		strTemp := strPath;
		strTemp := CONCAT(strTemp , aFileList[intOldestFile].sFileName);
		THIS^.M_FileDelete(strTemp);
		
		IF (uinSubStep = cSubStep_Finished) THEN
			intCmd := cFOLDER_HDL_CMD_DONE;
			uinStep := cStep_Refresh; 
		ELSIF (uinSubStep = cSubStep_Error) THEN
			intCmd := cFOLDER_HDL_CMD_DONE;
			uinStep := cStep_Error;
		END_IF
		
	cStep_Error:	
		// entry action
		IF (uinStep<>uinStep_old) THEN
			// written in sub Out_strInfo := 'Error';
			Out_bolBusy := FALSE;
			uinStep_old := uinStep;
		END_IF
		
		IF (intCmd<>cFOLDER_HDL_CMD_DONE) THEN
			Out_udiErrId := 0;
			uinSubStep := cSubStep_Done;
			uinStep := cStep_Wait4Job;
		END_IF
END_CASE

PROPERTY PUBLIC FileSupervisionPeriod : TIME
GET
FileSupervisionPeriod := timFileSupervisionPeriod;
END_GET
SET
timFileSupervisionPeriod := FileSupervisionPeriod;
END_SET
END_PROPERTY

PROPERTY PUBLIC get_FileList : ARRAY[1..cFILE_HDL_MAX_NR_OF_FILE_TO_MANAGE]  OF ST_FindFileEntry;
GET
uinSubStep := 0;

WHILE (THIS^.M_RefreshFileList()=FALSE) DO
	//wait until read all files in folder
END_WHILE

THIS^.M_SortFileList(); // sort last write date -> oldest at position 1!
END_GET
END_PROPERTY

PROPERTY get_NewestFileEntry : ST_FindFileEntry
GET
uinSubStep := 0;
(* läuft nicvht???
WHILE (THIS^.M_RefrehFileList()=FALSE) DO
	//wait until read all files in folder
END_WHILE

THIS^.M_SortFileList(); // sort last write date -> oldest at position 1!
*)
get_NewestFileEntry := aFileList[udiNrOfFilesInFolder];
END_GET
END_PROPERTY

METHOD PUBLIC M_Cmd_RefreshFileList : BOOL
intCmd := cFOLDER_HDL_CMD_REFRESH_FILE_LIST;
END_METHOD

METHOD PROTECTED M_FileDelete : BOOL
VAR_INPUT
	strPathName : T_MaxString;  
END_VAR
VAR
	strMyName : STRING := 'M_FileDelete: ';
END_VAR

CASE uinSubStep OF
	cSubStep_Done:	
		Out_strInfo :=  CONCAT(CONCAT(Out_strInfo, strMyName) , 'start');
		
		fbFileDelete_1.sNetId := strNetId;
		fbFileDelete_1.sPathName := strPathName;
		fbFileDelete_1.ePath := PATH_GENERIC;
		fbFileDelete_1.tTimeout := T#3S;
		fbFileDelete_1(bExecute:= FALSE);
		fbFileDelete_1(bExecute:= TRUE);
		
		uinSubStep := 1;
		
	1: 
		Out_strInfo :=  CONCAT(CONCAT(Out_strInfo, strMyName) , 'busy');	

		(* wait until function block not busy *)
		fbFileDelete_1( bExecute := FALSE );
		IF NOT fbFileDelete_1.bBusy THEN
			IF NOT fbFileDelete_1.bError THEN
				uinSubStep := cSubStep_Finished;
			ELSE 
				Out_udiErrId := fbFileDelete_1.nErrID;
				uinSubStep := cSubStep_Error;
			END_IF
		END_IF
		
	cSubStep_Finished: 
		// succesfully finished
		
	cSubStep_Error:
		Out_strInfo :=  CONCAT(CONCAT(Out_strInfo, strMyName) , CONCAT('error active - number:' , DWORD_TO_HEXSTR( fbFileDelete_1.nErrID, 0, FALSE )));
		Out_udiErrId := fbFileDelete_1.nErrID;
END_CASE
END_METHOD

METHOD PUBLIC M_FileExist : BOOL
VAR_INPUT
	strPathName : Tc2_System.T_MaxString;
END_VAR
VAR
	fbEnum : FB_EnumFindFileEntry := ( sNetID := '', tTimeout := T#5S, sPathName := strPathName );
	uinState : UINT:=0;
END_VAR
WHILE (uinState<>10) DO
	CASE uinState OF
	0:
		fbEnum.sNetId := strNetId;
		fbEnum.eCmd := eEnumCmd_First; (* enum first entry *)
		uinState := 1;
	
	1: (* enum one entry *)
		fbEnum( bExecute := FALSE );
		fbEnum( bExecute := TRUE );
		uinState := 2;
	
	2: (* wait until function block not busy *)
		fbEnum( bExecute := FALSE );
		IF NOT fbEnum.bBusy THEN
			IF NOT fbEnum.bError THEN
				IF NOT fbEnum.bEOE THEN
					M_FileExist := TRUE;
					EXIT;
				ELSE (* no more entries *)
					M_FileExist := FALSE;
					EXIT;
				END_IF
			ELSE (* log error *)
				M_FileExist := FALSE;
				EXIT;
			END_IF
		END_IF
	END_CASE
END_WHILE
END_METHOD

METHOD M_getFileInfo : ST_FindFileEntry
VAR_INPUT
	IN_strFileNameWithExt : Tc2_System.T_MaxString;// Contains the filename with extension
END_VAR
VAR
	ii : UDINT;
	udiUpperLimit : UDINT;
END_VAR
IF (udiNrOfFilesInFolder<cFILE_HDL_MAX_NR_OF_FILE_TO_MANAGE) THEN
	udiUpperLimit := udiNrOfFilesInFolder;
ELSE
	udiUpperLimit := cFILE_HDL_MAX_NR_OF_FILE_TO_MANAGE;	
END_IF

FOR ii:= 0 TO udiUpperLimit DO
	IF (FIND(aFileList[ii].sFileName,IN_strFileNameWithExt)<>0) THEN
		M_getFileInfo := aFileList[ii];
		EXIT;
	END_IF
END_FOR
END_METHOD

METHOD PUBLIC M_GetFileSize : LREAL
VAR_INPUT
	In_strFileName: T_MaxString;
END_VAR
VAR
	i:UDINT;
END_VAR
IF (udiNrOfFilesInFolder=0) THEN
	WHILE (THIS^.M_RefreshFileList()=FALSE) DO
		//wait until read all files in folder
	END_WHILE
END_IF

M_GetFileSize := 0.0;

FOR i := 1 TO udiNrOfFilesInFolder BY 1 DO
	IF (In_strFileName = aFileList[i].sFileName) THEN
		M_GetFileSize := Tc2_Utilities.UINT64_TO_LREAL(aFileList[i].fileSize);
		EXIT;
	END_IF
END_FOR;
END_METHOD

METHOD PUBLIC M_Init : BOOL
VAR_INPUT
	IN_strPath : Tc2_System.T_MaxString; 	// Contains only the path 
	IN_strPrefixFileName : Tc2_System.T_MaxString;// Contains only the filename
	IN_strFileExt : Tc2_System.T_MaxString;	// Contains only the ext
	In_strNetId: STRING(23); // NetId to write to foreign system drives
END_VAR
VAR
	strTemp: Tc2_System.T_MaxString;
END_VAR
strNetId := In_strNetId;
strPath := IN_strPath;
strFilePrefix := IN_strPrefixFileName;
strFileExt := IN_strFileExt;
strTemp := strPath;//todo check path allready added / CONCAT(strPath , '\');
strTemp := CONCAT(strTemp , strFilePrefix);
IF (strFileExt='') THEN
	strPathName := strTemp;
ELSE
	strTemp := CONCAT(strTemp , '.');
	strPathName := CONCAT(strTemp , strFileExt);
END_IF
uinStep := 0;
bolInitDone := TRUE;
END_METHOD

METHOD PUBLIC M_RefreshFileList : BOOL
VAR
	strMyName : STRING := 'M_RefrehFileList: ';
	strTemp : STRING;
END_VAR
CASE uinSubStep OF
	cSubStep_Done:	
		Out_strInfo :=  CONCAT(CONCAT(Out_strInfo, strMyName) , 'start');
		
		M_RefreshFileList := FALSE;
		udiNrOfFilesInFolder := 0;
		
		// define proberties for searching files in folder
		fbEnumFindFileList_1.sNetId := strNetId;

		strTemp := strPath;//todo check path allready added / CONCAT(strPath , '\');
		strTemp := CONCAT(strTemp , strFilePrefix);
		IF (strFileExt='') THEN
			strTemp := CONCAT(strTemp , '*'); // all data types
		ELSE
			strTemp := CONCAT(strTemp , '*.');
			strTemp := CONCAT(strTemp , strFileExt);
		END_IF

		fbEnumFindFileList_1.sPathName := strTemp; // read all files in the defined folder with the defined extension
        fbEnumFindFileList_1.pFindList := ADR(aFileList);
        fbEnumFindFileList_1.cbFindList := SIZEOF(aFileList);
        fbEnumFindFileList_1.tTimeout := DEFAULT_ADS_TIMEOUT;
		fbEnumFindFileList_1.eCmd := E_EnumCmdType.eEnumCmd_First;	(* enum first entry *)
		uinSubStep := 1;
		
	1: 
		Out_strInfo :=  CONCAT(CONCAT(Out_strInfo, strMyName) , 'Reading files in folder busy');	
		
		(* enum one entry *)
		IF bolAbort THEN
			bolAbort := FALSE;
			fbEnumFindFileList_1.eCmd := E_EnumCmdType.eEnumCmd_Abort;
		END_IF
		
		fbEnumFindFileList_1( bExecute := FALSE );
		fbEnumFindFileList_1( bExecute := TRUE );
		uinSubStep := 2;
		
	2:	
		Out_strInfo := CONCAT(CONCAT(Out_strInfo, strMyName) , 'Reading files in folder busy');	
		
		(* wait until function block not busy *)
		fbEnumFindFileList_1( bExecute := FALSE );
		IF NOT fbEnumFindFileList_1.bBusy THEN
			udiNrOfFilesInFolder := fbEnumFindFileList_1.nFindFiles;
			IF NOT fbEnumFindFileList_1.bError THEN
				IF NOT fbEnumFindFileList_1.bEOE THEN
					bolFileNrExceedArraySize := TRUE;
					(* read more informations -> not meaningful 
					fbEnumFindFileList_1.eCmd := E_EnumCmdType.eEnumCmd_Next; (* enum next entry *)
					uinSubStep := 1;*)
					uinSubStep := cSubStep_Finished; // reduce maximum in cyclic actions...-> delete if > max 
				ELSE (* no more entries *)
					uinSubStep := cSubStep_Finished;
				END_IF
			ELSE (* log error *)
				Out_udiErrId := fbEnumFindFileList_1.nErrID;
				uinSubStep := cSubStep_Error;
			END_IF
		END_IF

	cSubStep_Finished: 
		// succesfully finished
		M_RefreshFileList := TRUE;
	cSubStep_Error:
		Out_strInfo :=  CONCAT(CONCAT(Out_strInfo, strMyName) , CONCAT('error active - number:' , DWORD_TO_HEXSTR( fbEnumFindFileList_1.nErrID, 0, FALSE )));
		Out_udiErrId := fbEnumFindFileList_1.nErrID;
		M_RefreshFileList := TRUE;
END_CASE
END_METHOD

METHOD PUBLIC M_SortFileList : BOOL
VAR_INPUT

END_VAR
VAR
	stTempFile 	: ST_FindFileEntry;
	bolNoChangeDone: BOOL;
	i,j :UDINT;
END_VAR
// BubbleSort
M_SortFileList := FALSE;

IF (udiNrOfFilesInFolder>1) THEN
	lreTotalFileSize := UINT64_TO_LREAL(aFileList[1].fileSize);
	FOR i := 1 TO udiNrOfFilesInFolder BY 1 DO
		bolNoChangeDone := TRUE;
		FOR j := 1 TO (udiNrOfFilesInFolder-i) BY 1 DO
			IF (i=1) THEN// count total filesize
				lreTotalFileSize := lreTotalFileSize + Tc2_Utilities.UINT64_TO_LREAL(aFileList[j+1].fileSize);
			END_IF
			
			IF (FILETIME_TO_DT(aFileList[j].lastWriteTime) > FILETIME_TO_DT(aFileList[j + 1].lastWriteTime)) THEN
				// swap files
				memcpy(ADR(stTempFile), ADR(aFileList[j]),SIZEOF(stTempFile));
				memcpy(ADR(aFileList[j]), ADR(aFileList[j + 1]),SIZEOF(stTempFile));
				memcpy(ADR(aFileList[j + 1]), ADR(stTempFile),SIZEOF(stTempFile));
				bolNoChangeDone := FALSE; // at least one change done
			END_IF
			
		END_FOR; 
		IF (bolNoChangeDone) THEN
			EXIT;
		END_IF
	END_FOR;
END_IF;
M_SortFileList := TRUE;
END_METHOD

PROPERTY MaxNrOfFilesInFolder : UINT
GET
MaxNrOfFilesInFolder := uinMaxNrOfFilesInFolder;
END_GET
SET
// not more files allowed as defined in struct....Sort problem
IF (MaxNrOfFilesInFolder<cFILE_HDL_MAX_NR_OF_FILE_TO_MANAGE) THEN
	uinMaxNrOfFilesInFolder := MaxNrOfFilesInFolder;
ELSE
	uinMaxNrOfFilesInFolder := UDINT_TO_UINT(cFILE_HDL_MAX_NR_OF_FILE_TO_MANAGE-1);	
END_IF
END_SET
END_PROPERTY

END_FUNCTION_BLOCK

// POUs/Utility/GHT [Generic Hash Table]/FB_GHT
FUNCTION_BLOCK FB_GHT IMPLEMENTS IGHT
VAR CONSTANT
	MAX_HASH_LISTS: INT := 3;
	MAX_HASHLIST_ENTRIES: INT := 50;
	CUTOFF_A: ULINT := 4000000000;
	CUTOFF_B: ULINT := 8000000000;
END_VAR
VAR
	m_bolDeleteItems: BOOL;
	m_uintCount: UINT;
	m_fbHashTable: ARRAY[0..(MAX_HASH_LISTS - 1)] OF FB_HashTableCtrl;
	m_hHashTable: ARRAY[0..(MAX_HASH_LISTS - 1)] OF T_HHASHTABLE;
	m_uliCutoff: ARRAY[0..(MAX_HASH_LISTS - 1)] OF ULINT;
	m_aHashTableBuffer: ARRAY[0..(MAX_HASH_LISTS - 1)] OF T_GHTHashTableBuffer;
END_VAR

{attribute 'object_name' := 'AddItem'}
METHOD AddItem : BOOL
VAR_INPUT
	uliKey: ULINT;
	pData: POINTER TO BYTE;
END_VAR
VAR
	iIdx: INT;
END_VAR
iIdx := GetTableIdx(uliKey);

m_fbHashTable[iIdx].A_Add( key := ULINT_TO_UDINT(uliKey-m_uliCutoff[iIdx]), putValue := pData, hTable := m_hHashTable[iIdx] );

IF m_fbHashTable[iIdx].bOk THEN
	m_uintCount := m_uintCount + 1;
END_IF
END_METHOD

{attribute 'object_name' := 'Clear'}
METHOD Clear : BOOL
VAR_INPUT
	bolFreePointer: BOOL;
END_VAR
VAR
	iIdx: INT;
	pData: POINTER TO BYTE;
END_VAR
FOR iIdx := 0 TO MAX_HASH_LISTS - 1 DO
	IF bolFreePointer THEN
		m_fbHashTable[iIdx].A_GetFirst(hTable := m_hHashTable[iIdx]);

		WHILE m_fbHashTable[iIdx].bOk DO
			pData := m_fbHashTable[iIdx].getValue;
			__DELETE(pData);
			m_fbHashTable[iIdx].A_GetNext(hTable := m_hHashTable[iIdx]);
		END_WHILE
		
	END_IF
	
	m_fbHashTable[iIdx].A_RemoveAll(hTable := m_hHashTable[iIdx]);
END_FOR

m_uintCount := 0;
END_METHOD

PROPERTY Count : UINT
GET
END_GET
END_PROPERTY

{attribute 'object_name' := 'FB_init'}
METHOD FB_init : BOOL
VAR_INPUT
	/// if TRUE, the retain variables are initialized (warm start / cold start)
	bInitRetains: BOOL;
	/// if TRUE, the instance afterwards gets moved into the copy code (online change)
	bInCopyCode: BOOL;
END_VAR
m_uliCutoff[0] := 0;
m_uliCutoff[1] := CUTOFF_A;
m_uliCutoff[2] := CUTOFF_B;

m_uintCount := 0;
END_METHOD

{attribute 'object_name' := 'GetTableIdx'}
METHOD PRIVATE GetTableIdx : INT
VAR_INPUT
	uliBarcode: ULINT;
END_VAR
IF uliBarcode < CUTOFF_A THEN
	GetTableIdx := 0;
	RETURN;
END_IF

IF uliBarcode > CUTOFF_B THEN
	GetTableIdx := 2;
	RETURN;
END_IF

GetTableIdx := 1;
END_METHOD

{attribute 'object_name' := 'Initialize'}
METHOD Initialize : BOOL
F_CreateHashTableHnd( ADR( m_aHashTableBuffer[0].aBuffer ), SIZEOF( m_aHashTableBuffer[0].aBuffer ), m_hHashTable[0] );
F_CreateHashTableHnd( ADR( m_aHashTableBuffer[1].aBuffer ), SIZEOF( m_aHashTableBuffer[1].aBuffer ), m_hHashTable[1] );
F_CreateHashTableHnd( ADR( m_aHashTableBuffer[2].aBuffer ), SIZEOF( m_aHashTableBuffer[2].aBuffer ), m_hHashTable[2] );
END_METHOD

{attribute 'object_name' := 'Lookup'}
METHOD Lookup : POINTER TO BYTE
VAR_INPUT
	uliKey: ULINT;
	bolRemove: BOOL;
END_VAR
VAR
	pfbHashTable: POINTER TO FB_HashTableCtrl;
	phHashTable: POINTER TO T_HHASHTABLE;
	uliCutoff: ULINT;
	iIdx: INT;
END_VAR
iIdx := GetTableIdx(uliKey);

m_fbHashTable[iIdx].A_Lookup( key := ULINT_TO_UDINT(uliKey-m_uliCutoff[iIdx]), hTable := m_hHashTable[iIdx] );

IF m_fbHashTable[iIdx].bOk THEN
	Lookup := m_fbHashTable[iIdx].getValue;
	
	IF bolRemove THEN
		m_fbHashTable[iIdx].A_Remove( key := ULINT_TO_UDINT(uliKey-m_uliCutoff[iIdx]), hTable := m_hHashTable[iIdx]);

		IF m_fbHashTable[iIdx].bOk THEN
			m_uintCount := m_uintCount - 1;
		END_IF
	END_IF
ELSE
	Lookup := NULL;
END_IF
END_METHOD

END_FUNCTION_BLOCK

// POUs/Utility/GHT [Generic Hash Table]/IGHT
INTERFACE IGHT

{attribute 'object_name' := 'AddItem'}
METHOD AddItem : BOOL
VAR_INPUT
	uliKey: ULINT;
	pData: POINTER TO BYTE;
END_VAR
END_METHOD

{attribute 'object_name' := 'Clear'}
METHOD Clear : BOOL
VAR_INPUT
	bolFreePointer: BOOL;
END_VAR
END_METHOD

PROPERTY Count : UINT
GET
END_GET
END_PROPERTY

{attribute 'object_name' := 'Initialize'}
METHOD Initialize : BOOL
END_METHOD

{attribute 'object_name' := 'Lookup'}
METHOD Lookup : POINTER TO BYTE
VAR_INPUT
	uliKey: ULINT;
	bolRemove: BOOL;
END_VAR
END_METHOD

END_INTERFACE

// POUs/Utility/Logger/BasLog/FB_BasLogTest_Client
FUNCTION_BLOCK FB_BasLogTest_Client
VAR_INPUT
	In_p_fbBasLog: POINTER TO FB_BasLog; // only one central FB_BasLog instance allowed per PLC!!!
END_VAR
VAR_OUTPUT
END_VAR
VAR
	stData : T_Bl_BaseStruc;
	bolInit : BOOL := FALSE;
	pReadHandle : POINTER TO POINTER TO T_Queue_Info;
	uinInitStatus : UINT;
	uinChangeMaskStatus :UINT;
	uinReadStatus : UINT;
	bolChangeMask : BOOL;
	bolRead : BOOL;
	fbTimeStamp: FB_TimeStamp;
END_VAR

(*__________________________________________________________________________________________________
¦	
¦	Vistaprint Schweiz GmbH
¦	CH - 8401 Winterthur
¦
¦	www.vistaprint.ch - info@vistaprint.ch
¦___________________________________________________________________________________________________

Function desription:
Example and test programm for testing the base log system - read data from base log

History:
Version		Date			Author		Comment
---------------------------------------------------------------------------------------------------
0.00.1		14.07.2014		AVME/KVO	Start history
___________________________________________________________________________________________________*)

// system init onetime after start up
IF (bolInit=FALSE) THEN
	// init timer system
	fbTimeStamp.In_strNetId := ''; // use local system time
	fbTimeStamp.In_t_CycleTimeRefreshTimeZone := T#15M; // cyclic check time zone settings
	//init baselog system, one time should be called per baslog system
	In_p_fbBasLog^.M_ClientInit(In_strClientName:='BaseLog',In_udiMask := 16#FFFFFFFF, In_uinNrOfElement:= 128,In_p_fbTimeStamp:=ADR(fbTimeStamp),In_bolUseLocalTimeStamp:=TRUE,Out_pHandle=>pReadHandle,Out_uinStatus=>uinInitStatus);
	
	bolInit := TRUE;
END_IF

fbTimeStamp(); // cyclic call needed for valid time stamp / synchronisation
	
(* change mak on runtime *)
IF (bolRead = TRUE) THEN
	(* cyclically read out of data*)
	uinReadStatus:= In_p_fbBasLog^.M_Read(In_pHandle:=pReadHandle,In_pData:=ADR(stData)); 
END_IF

(* change mask on runtime *)
IF (bolChangeMask = TRUE) THEN
	uinChangeMaskStatus := In_p_fbBasLog^.M_ChangeMask(In_strClientName:='BaseLog',In_udiNewMask:= 16#0F0F0F0F);
	bolChangeMask := FALSE;
END_IF

END_FUNCTION_BLOCK

// POUs/Utility/Logger/BasLog/FB_BasLogTest_Sender
FUNCTION_BLOCK FB_BasLogTest_Sender
VAR_INPUT
	In_p_fbBasLog: POINTER TO FB_BasLog; // only one central FB_BasLog instance allowed per PLC!!!
END_VAR
VAR_OUTPUT
END_VAR
VAR
	bolInit : BOOL := FALSE;
	pHandle : POINTER TO T_Bl_LibHandleRow;
	uinGetHandleStatus : UINT;
	uinWriteStatus :UINT;
	uinDoWrite : UINT;
	dinPar1 : DINT;
	strText1 : STRING(30):='Controller 1';
	strText2 : STRING(30):='Alarm sub info';
END_VAR

(*__________________________________________________________________________________________________
¦	
¦	Vistaprint Schweiz GmbH
¦	CH - 8401 Winterthur
¦
¦	www.vistaprint.ch - info@vistaprint.ch
¦___________________________________________________________________________________________________

Function desription:
Example and test programm for testing the queue system - write data to base log

History:
Version		Date			Author		Comment
---------------------------------------------------------------------------------------------------
0.00.1		14.07.2014		AVME/KVO	Start history
___________________________________________________________________________________________________*)

// system init onetime after start up
IF (bolInit=FALSE) THEN
	uinGetHandleStatus := In_p_fbBasLog^.M_GetHandle(Out_pHandle=>pHandle);
	
	bolInit := TRUE;
END_IF

// write base log entries
IF (uinDoWrite>0) THEN
	uinDoWrite := uinDoWrite - 1;
	dinPar1 := dinPar1 + 1;
	uinWriteStatus := In_p_fbBasLog^.M_Log(In_pHandle:=pHandle,In_udiLogType:=BasLog.cLOGTYPE_ALARM,In_intCtrlID:=11,In_strText1:=strText1,In_strText2:=strText2,In_dinPar1:=dinPar1,In_dinPar2:=0,In_dinPar3:=0,In_dinPar4:=0) ;
END_IF

END_FUNCTION_BLOCK

// POUs/Utility/Logger/DatLog/FB_DatLog
FUNCTION_BLOCK FB_DatLog
VAR_INPUT
END_VAR
VAR_OUTPUT
END_VAR
VAR
	stDatLogLibInfo : T_DL_LibInfo;
	fbPLC_ReadSymInfo: PLC_ReadSymInfoByNameEx; // only one init allowed on the same time....
END_VAR

(*__________________________________________________________________________________________________
¦	
¦	Vistaprint Schweiz GmbH
¦	CH - 8401 Winterthur
¦
¦	www.vistaprint.ch - info@vistaprint.ch
¦___________________________________________________________________________________________________

Function desription:
Base logger system. The FUB must be called defined globally one time in PLC-program. After that the implemented 
sender and receiver must interact over the public methodes of the FB_BasLog.

History:
Version		Date			Author		Comment
---------------------------------------------------------------------------------------------------
0.00.1		14.07.2014		AVME/KVO	Start history
___________________________________________________________________________________________________*)

METHOD PROTECTED M_AllocMEM : POINTER TO BYTE

VAR_INPUT
	In_SizeOfBuffer : UINT; // Byte size of quee to allocate
END_VAR
// Debug counter
M_AllocMEM := __NEW(BYTE,In_SizeOfBuffer);

// check if allocate memory is ok
IF (M_AllocMEM=TC3_MEMMAN.NULL) THEN
	M_AllocMEM := TC3_MEMMAN.NULL;
ELSE
	Tc2_System.MEMSET(M_AllocMEM,0,In_SizeOfBuffer); // init with zero.
END_IF
END_METHOD

METHOD PRIVATE M_CheckAndAppendDatLogInfo : Pointer TO T_DL_SysInfo
VAR_INPUT
	In_strDatLogName: STRING(DatLog.cMAX_SYS_NAME_LENGTH); // name of the client
END_VAR
VAR
	pstSysInfo: POINTER TO T_DL_SysInfo;
END_VAR
// methode check, if data log allready exists and if not allocate a new system
// -> return reference on new system

// exist at least one data log system
IF (stDatLogLibInfo.pstDatLogSysInfo=TC3_MEMMAN.NULL) THEN
	// create  a new system
	stDatLogLibInfo.pstDatLogSysInfo := M_AllocMEM(SIZEOF(T_DL_SysInfo));

	IF (stDatLogLibInfo.pstDatLogSysInfo=TC3_MEMMAN.NULL) THEN
		M_CheckAndAppendDatLogInfo := TC3_MEMMAN.NULL;
		RETURN;
	END_IF
	
	// data log name entry in info system
	stDatLogLibInfo.pstDatLogSysInfo^.strDatLogName := In_strDatLogName;
	M_CheckAndAppendDatLogInfo := stDatLogLibInfo.pstDatLogSysInfo;
	RETURN;
END_IF

// after this point the system has to exist
IF (stDatLogLibInfo.pstDatLogSysInfo<>TC3_MEMMAN.NULL) THEN
	pstSysInfo := stDatLogLibInfo.pstDatLogSysInfo;
	
	WHILE (pstSysInfo<>TC3_MEMMAN.NULL) DO
		IF (pstSysInfo^.strDatLogName=In_strDatLogName) THEN
			// data log name found -> return handle
			M_CheckAndAppendDatLogInfo := pstSysInfo;
			RETURN;
		END_IF
		
		// last element
		IF (pstSysInfo^.pstNextDatLogSystem=TC3_MEMMAN.NULL) THEN
			// the requested log name does not exist -> allocate a new one
			pstSysInfo^.pstNextDatLogSystem := M_AllocMEM(SIZEOF(T_DL_SysInfo));

			IF (pstSysInfo^.pstNextDatLogSystem<>TC3_MEMMAN.NULL) THEN
				pstSysInfo := pstSysInfo^.pstNextDatLogSystem;
				// data log name entry in info system
				pstSysInfo^.strDatLogName := In_strDatLogName;
				M_CheckAndAppendDatLogInfo := pstSysInfo;
				RETURN;
			ELSE
				M_CheckAndAppendDatLogInfo := TC3_MEMMAN.NULL;
				RETURN;
			END_IF
		ELSE
			// reference next
			pstSysInfo := pstSysInfo^.pstNextDatLogSystem;
		END_IF
	END_WHILE
END_IF
END_METHOD

METHOD PUBLIC M_GetHandle : UINT
VAR_INPUT
	In_strDatLogName: STRING(DatLog.cMAX_SYS_NAME_LENGTH); // name of the client
	In_p_fbBasLog: POINTER TO FB_BasLog; // only one central FB_BasLog instance allowed per PLC!!!
END_VAR
VAR_OUTPUT
	Out_pHandle : POINTER TO BYTE; // handle of log system for write (M_Log)
	Out_udiStatus : UDINT; //0 => successful done, <>0 => error
END_VAR
VAR
	pstSysInfo: POINTER TO T_DL_SysInfo;
	uinGetHandleStatus : UINT;
END_VAR

// check if log system allready exists or not, if not allocate a new one
	pstSysInfo := M_CheckAndAppendDatLogInfo(In_strDatLogName:=In_strDatLogName);
	IF (pstSysInfo=TC3_MEMMAN.NULL) THEN
		Out_udiStatus := DatLog.cERR_MEM_ALLOC;
		RETURN;
	END_IF
	
	// log on base log system
	uinGetHandleStatus := In_p_fbBasLog^.M_GetHandle(Out_pHandle=>pstSysInfo^.pBaseLogHandle);
	
	// check error
	IF (uinGetHandleStatus<>0) THEN
		Out_udiStatus := UINT_TO_UDINT(uinGetHandleStatus);
		RETURN;
	ELSE
		pstSysInfo^.p_fbBasLog := In_p_fbBasLog;
		Out_pHandle := pstSysInfo;
	END_IF
END_METHOD

METHOD PUBLIC M_Init : BOOL
VAR_INPUT
	In_bolExecute : BOOL;
	In_strDatLogName: STRING(DatLog.cMAX_SYS_NAME_LENGTH); // name of the client
	In_a_strDataDefinition: ARRAY[0..DatLog.cMAX_NR_OF_VAR] OF STRING(DatLog.cMAX_VAR_NAME_LEN); // complete VarName: p.e.:MAIN.INIT_TASK.VARINT
	In_uinStartId: UINT;	// Start ident for item index -> cfg file config has to match with this number!
	In_Port : T_AmsPort;	// on plc the first runtime system is the 801, 811 ...
END_VAR
VAR_OUTPUT
	Out_udiStatus: UDINT;		 // 0 => successful done, <>0 => error
	Out_bolDone: BOOL;			// Done
END_VAR
VAR
	pstSysInfo: POINTER TO T_DL_SysInfo;
	pstItem : POINTER TO T_DL_Item;
	ii : UINT;
END_VAR

IF (In_bolExecute=TRUE) THEN
	// check if log system allready exists or not, if not allocate a new one
	pstSysInfo := M_CheckAndAppendDatLogInfo(In_strDatLogName:=In_strDatLogName);
	IF (pstSysInfo=TC3_MEMMAN.NULL) THEN
		Out_udiStatus := DatLog.cERR_MEM_ALLOC;
		RETURN;
	END_IF

	IF (stDatLogLibInfo.stStatemachine.bolExecute_old=FALSE) THEN // reset statemachine
		stDatLogLibInfo.stStatemachine.uinState := 1;
		Out_bolDone := FALSE;
		Out_udiStatus := 0;
		stDatLogLibInfo.stStatemachine.usiInitDone := 0;
	END_IF

CASE stDatLogLibInfo.stStatemachine.uinState OF
	1:
		//check number of elements
		FOR ii :=0 TO DatLog.cMAX_NR_OF_VAR BY 1 DO
			IF (In_a_strDataDefinition[ii]='') THEN
				EXIT;
			END_IF
		END_FOR
		
		pstSysInfo^.uinNbrOfItems := ii;
		pstSysInfo^.uinStartId := In_uinStartId;
		
		// allocate memory for items
		pstSysInfo^.pstItems := M_AllocMEM((pstSysInfo^.uinNbrOfItems*SIZEOF(T_DL_Item)));
		IF (pstSysInfo^.pstItems =TC3_MEMMAN.NULL) THEN
			Out_udiStatus := DatLog.cERR_MEM_ALLOC;
			RETURN;
		END_IF
		pstSysInfo^.uinCntReadItems := 0;
		pstSysInfo^.uinItemOffset := 0;
		stDatLogLibInfo.stStatemachine.uinState := stDatLogLibInfo.stStatemachine.uinState + 1;
		
	2:	
		fbPLC_ReadSymInfo.NETID:=''; // local PLC
		IF (In_Port=0) THEN// access first runtime system
			fbPLC_ReadSymInfo.PORT := 851;
		ELSE
			fbPLC_ReadSymInfo.PORT := In_Port;
		END_IF
		fbPLC_ReadSymInfo.SYMNAME := In_a_strDataDefinition[pstSysInfo^.uinCntReadItems];
		fbPLC_ReadSymInfo.START := FALSE;
		fbPLC_ReadSymInfo();
		fbPLC_ReadSymInfo.START := TRUE;
		fbPLC_ReadSymInfo();
		stDatLogLibInfo.stStatemachine.uinState := stDatLogLibInfo.stStatemachine.uinState + 1;
		
	3:
		fbPLC_ReadSymInfo();
		IF (fbPLC_ReadSymInfo.BUSY=FALSE) THEN
			stDatLogLibInfo.stStatemachine.uinState := stDatLogLibInfo.stStatemachine.uinState + 1;
		END_IF
		
	4:
		pstItem := pstSysInfo^.pstItems;
		IF (fbPLC_ReadSymInfo.ERR=FALSE) THEN
			pstItem[pstSysInfo^.uinCntReadItems].strPvName := In_a_strDataDefinition[pstSysInfo^.uinCntReadItems];
			pstItem[pstSysInfo^.uinCntReadItems].uinItemOffset := pstSysInfo^.uinItemOffset;
			pstItem[pstSysInfo^.uinCntReadItems].SymInfo := fbPLC_ReadSymInfo.SYMINFO;
			pstSysInfo^.uinItemOffset := pstSysInfo^.uinItemOffset + UDINT_TO_UINT(pstItem[pstSysInfo^.uinCntReadItems].SymInfo.byteSize); // offset for next
			
			// check if type ok/allowed
			IF (pstItem[pstSysInfo^.uinCntReadItems].SymInfo.symDataType = 'BOOL') THEN 
				pstItem[pstSysInfo^.uinCntReadItems].udiItemType := DatLog.cVAR_TYPE_BOOL;
			ELSIF (pstItem[pstSysInfo^.uinCntReadItems].SymInfo.symDataType = 'SINT') THEN 
				pstItem[pstSysInfo^.uinCntReadItems].udiItemType := DatLog.cVAR_TYPE_SINT;
			ELSIF (pstItem[pstSysInfo^.uinCntReadItems].SymInfo.symDataType = 'INT') THEN 
				pstItem[pstSysInfo^.uinCntReadItems].udiItemType := DatLog.cVAR_TYPE_INT;
			ELSIF (pstItem[pstSysInfo^.uinCntReadItems].SymInfo.symDataType = 'DINT') THEN 
				pstItem[pstSysInfo^.uinCntReadItems].udiItemType := DatLog.cVAR_TYPE_DINT;
			ELSIF (pstItem[pstSysInfo^.uinCntReadItems].SymInfo.symDataType = 'USINT') THEN 
				pstItem[pstSysInfo^.uinCntReadItems].udiItemType := DatLog.cVAR_TYPE_USINT;
			ELSIF (pstItem[pstSysInfo^.uinCntReadItems].SymInfo.symDataType = 'UINT') THEN 
				pstItem[pstSysInfo^.uinCntReadItems].udiItemType := DatLog.cVAR_TYPE_INT;
			ELSIF (pstItem[pstSysInfo^.uinCntReadItems].SymInfo.symDataType = 'UDINT') THEN 
				pstItem[pstSysInfo^.uinCntReadItems].udiItemType := DatLog.cVAR_TYPE_UDINT;
			ELSIF (pstItem[pstSysInfo^.uinCntReadItems].SymInfo.symDataType = 'REAL') THEN 
				pstItem[pstSysInfo^.uinCntReadItems].udiItemType := DatLog.cVAR_TYPE_REAL;
			ELSIF (FIND(STR1:=pstItem[pstSysInfo^.uinCntReadItems].SymInfo.symDataType,STR2:='STRING')<>0) THEN 
				IF (pstItem[pstSysInfo^.uinCntReadItems].SymInfo.byteSize < BasLog.cMAX_CHAR_TEXT2) THEN
					pstItem[pstSysInfo^.uinCntReadItems].udiItemType := DatLog.cVAR_TYPE_STRING;
				ELSE
					Out_udiStatus := DatLog.cERR_UNSUPPORTED_TYPE_STRING_TOO_LONG;
					RETURN;
				END_IF
			ELSE
				Out_udiStatus := DatLog.cERR_UNSUPPORTED_TYPE;
				RETURN;
			END_IF
		ELSE
			Out_udiStatus := fbPLC_ReadSymInfo.ERRID;
			RETURN;
		END_IF
		
		pstSysInfo^.uinCntReadItems := pstSysInfo^.uinCntReadItems  + 1;
		IF (pstSysInfo^.uinCntReadItems<pstSysInfo^.uinNbrOfItems) THEN // read next value
			stDatLogLibInfo.stStatemachine.uinState := 2;
		ELSE
			stDatLogLibInfo.stStatemachine.uinState := stDatLogLibInfo.stStatemachine.uinState + 1; // all items found
		END_IF
	5:
		Out_bolDone := TRUE;
		Out_udiStatus := 0;
		pstSysInfo^.usiInitOk := 1; 
END_CASE
END_IF
stDatLogLibInfo.stStatemachine.bolExecute_old := In_bolExecute;
END_METHOD

METHOD PUBLIC M_Log : UINT
VAR_INPUT
	In_pHandle : POINTER TO BYTE;// handle of log system for write (M_Log)
	In_a_pData: ARRAY [0..DatLog.cMAX_NR_OF_VAR] OF POINTER TO BYTE;// address of structure elements
END_VAR
VAR_OUTPUT
	Out_udiStatus: UDINT;		// 0 => successful done, <>0 => error
END_VAR
VAR
	pstSysInfo: POINTER TO T_DL_SysInfo;
	pstItem : POINTER TO T_DL_Item;
	pstItemEle : T_DL_Item;
	ii : UINT;
	strText2: STRING(BasLog.cMAX_CHAR_TEXT2); // informationtext2
	dinPar2 : DINT;
	dinId : DINT;
	uinStatus : UINT;
END_VAR
// check handle ok
IF (In_pHandle=TC3_MEMMAN.NULL) THEN
	M_Log := DatLog.cERR_NO_HANDLE;
	RETURN;
END_IF

// check data
IF (In_a_pData[0]=TC3_MEMMAN.NULL) THEN
	M_Log := DatLog.cERR_NO_DATE;
	RETURN;
END_IF

// access data loggger system info
pstSysInfo := In_pHandle;

// check if init ok
IF (pstSysInfo^.usiInitOk=0) THEN
	M_Log := DatLog.cERR_INIT_FAILED;
	RETURN;
END_IF

// check if items
IF (pstSysInfo^.pstItems=TC3_MEMMAN.NULL) OR (pstSysInfo^.uinNbrOfItems<=0) THEN
	M_Log := DatLog.cERR_NO_ITEMS;
	RETURN;
END_IF
// access item definitions
pstItem := pstSysInfo^.pstItems;

// inc. record id: important the id is inc bevor and after writing of data -> to be sure that no second write is done (MUTEX)
stDatLogLibInfo.udiCommonRecIdx := stDatLogLibInfo.udiCommonRecIdx + 1;
IF (stDatLogLibInfo.udiCommonRecIdx=0) THEN
	stDatLogLibInfo.udiCommonRecIdx := stDatLogLibInfo.udiCommonRecIdx + 1;
END_IF
// write record start
// AE_BL_VAR_TYPE_CMD_NEW_REC
uinStatus := pstSysInfo^.p_fbBasLog^.M_Log(In_pHandle := pstSysInfo^.pBaseLogHandle,In_udiLogType:=BasLog.cLOGTYPE_DATA,In_intCtrlID:=DatLog.cCTRL_ID,In_strText1:='DataLog',In_strText2:='AE_BL_VAR_TYPE_CMD_NEW_REC',In_dinPar1:=0,In_dinPar2:=0,In_dinPar3:=BasLog.cVAR_TYPE_CMD_NEW_REC,In_dinPar4:=UDINT_TO_DINT(stDatLogLibInfo.udiCommonRecIdx));
IF (uinStatus<>0) THEN
	M_Log := uinStatus;
	RETURN;
END_IF

// loop over all items and write data to logger
FOR ii :=0 TO (pstSysInfo^.uinNbrOfItems-1) BY 1 DO
	// write item
	pstItemEle := pstItem[ii]; // for debugging
	// id
	dinId := UINT_TO_DINT(pstSysInfo^.uinStartId + ii);
	IF (pstItem[ii].udiItemType=DatLog.cVAR_TYPE_STRING) THEN
		MEMSET(destAddr:=ADR(strText2),fillByte:=0,n:= SIZEOF(strText2)); // to be sure that a zero is at the end
		// doesn't work with beckhoff...MEMCPY(destAddr := ADR(strText2),srcAddr:= (In_pAdrData + pstItem[ii].uinItemOffset),n:=pstItem[ii].SymInfo.byteSize);
		MEMCPY(destAddr := ADR(strText2),srcAddr:= In_a_pData[ii],n:=pstItem[ii].SymInfo.byteSize);
		dinPar2 := 0;
	ELSE
		strText2 := pstItem[ii].strPvName; // just for info
		MEMCPY(destAddr := ADR(dinPar2),srcAddr:= In_a_pData[ii],n:=pstItem[ii].SymInfo.byteSize);
	END_IF
	
	// log item
	uinStatus := pstSysInfo^.p_fbBasLog^.M_Log(In_pHandle := pstSysInfo^.pBaseLogHandle,In_udiLogType:=BasLog.cLOGTYPE_DATA,In_intCtrlID:=DatLog.cCTRL_ID,In_strText1:='DataLog',In_strText2:=strText2,In_dinPar1:=dinId,In_dinPar2:=dinPar2,In_dinPar3:=UDINT_TO_DINT(pstItem[ii].udiItemType),In_dinPar4:=UDINT_TO_DINT(stDatLogLibInfo.udiCommonRecIdx));

	IF (uinStatus<>0) THEN // no stop write error number
		M_Log := uinStatus;
	END_IF
END_FOR

// write record stop
// AE_BL_VAR_TYPE_CMD_NEW_REC
uinStatus := pstSysInfo^.p_fbBasLog^.M_Log(In_pHandle := pstSysInfo^.pBaseLogHandle,In_udiLogType:=BasLog.cLOGTYPE_DATA,In_intCtrlID:=DatLog.cCTRL_ID,In_strText1:='DataLog',In_strText2:='AE_BL_VAR_TYPE_CMD_END_REC',In_dinPar1:=0,In_dinPar2:=0,In_dinPar3:=BasLog.cVAR_TYPE_CMD_END_REC,In_dinPar4:=UDINT_TO_DINT(stDatLogLibInfo.udiCommonRecIdx));
IF (uinStatus<>0) THEN
	M_Log := uinStatus;
	RETURN;
END_IF

// increment id a second time
stDatLogLibInfo.udiCommonRecIdx := stDatLogLibInfo.udiCommonRecIdx + 1;
IF (stDatLogLibInfo.udiCommonRecIdx=0) THEN
	stDatLogLibInfo.udiCommonRecIdx := stDatLogLibInfo.udiCommonRecIdx + 1;
END_IF
END_METHOD

END_FUNCTION_BLOCK

// POUs/Utility/Logger/DatLog/FB_DatLogTest_Sender
FUNCTION_BLOCK FB_DatLogTest_Sender
VAR_INPUT
	In_p_fbBasLog: POINTER TO FB_BasLog; // only one central FB_BasLog instance allowed per PLC!!!
	In_a_pData: ARRAY [0..DatLog.cMAX_NR_OF_VAR] OF POINTER TO BYTE;
	In_strTaskName: STRING(20);
	In_strValueNameOfData: STRING(20);
END_VAR
VAR_OUTPUT
	Out_bolInit : BOOL := FALSE;
END_VAR
VAR
	bolDone : BOOL;
	pDL_Handle: POINTER TO T_DL_SysInfo;
	udiStatusInit :UDINT;
	udiStatus : UDINT;
	fbDatLog: FB_DatLog;
	a_strDataDefinition :ARRAY[0..DatLog.cMAX_NR_OF_VAR] OF STRING(DatLog.cMAX_VAR_NAME_LEN);
	uinDoLogData : UINT;
	strTemp: T_MaxString;
	strTemp2: T_MaxString;
	ii : UINT;
END_VAR

(*__________________________________________________________________________________________________
¦	
¦	Vistaprint Schweiz GmbH
¦	CH - 8401 Winterthur
¦
¦	www.vistaprint.ch - info@vistaprint.ch
¦___________________________________________________________________________________________________

Function desription:
Example and test programm for testing the data logger system - write data to data log

History:
Version		Date			Author		Comment
---------------------------------------------------------------------------------------------------
0.00.1		02.09.2014		AVME/KVO	Start history
___________________________________________________________________________________________________*)

// system init onetime after start up
IF (Out_bolInit=FALSE) THEN
	
	// TODO :parse a struct on PLC...
	FOR ii := 0 TO DatLog.cMAX_NR_OF_VAR DO
		strTemp := In_strTaskName;
		strTemp := CONCAT(STR1 := strTemp,'.');
		strTemp := CONCAT(STR1 := strTemp,In_strValueNameOfData);
		strTemp := CONCAT(STR1 := strTemp,'.');
		// fillup variable elements of struct, order is important!!!!!!!!!!!!!!!!!!!!
		CASE ii OF
			0:
				strTemp2 := 'bolOk';
			1:
				strTemp2 := 'intCnt';
			2:
				strTemp2 := 'strNewText';
		ELSE
			EXIT;
		END_CASE
		a_strDataDefinition[ii] := CONCAT(STR1 := strTemp,STR2:=strTemp2);
	END_FOR
	
	fbDatLog.M_Init(In_bolExecute := TRUE,In_strDatLogName:= 'DatLog',In_a_strDataDefinition:=a_strDataDefinition,In_Port:=851,In_uinStartId:=100,Out_udiStatus=>udiStatusInit,Out_bolDone=>bolDone);
	IF (bolDone OR (udiStatusInit<>0)) THEN
		fbDatLog.M_Init(In_bolExecute := FALSE,In_strDatLogName:= 'DatLog',In_a_strDataDefinition:=a_strDataDefinition,In_Port:=851,In_uinStartId:=100); // reset statemachine
	
		IF (udiStatusInit=0) THEN
			udiStatusInit := fbDatLog.M_GetHandle(In_strDatLogName:='DatLog',In_p_fbBasLog:=In_p_fbBasLog,Out_pHandle=>pDL_Handle,Out_udiStatus=>udiStatusInit);
		END_IF
		
		Out_bolInit := TRUE;
	END_IF

ELSE
	fbDatLog.M_Init(In_bolExecute := FALSE,In_strDatLogName:= 'DatLog',In_a_strDataDefinition:=a_strDataDefinition,In_Port:=851,In_uinStartId:=100); // reset statemachine
	
END_IF

// write entry data 
IF ((pDL_Handle<>TC3_MEMMAN.NULL) AND (udiStatusInit=0) AND (Out_bolInit=TRUE)) THEN
	fbDatLog.M_Log(In_pHandle:=pDL_Handle,In_a_pData:= In_a_pData,Out_udiStatus=>udiStatus);
END_IF

END_FUNCTION_BLOCK

// POUs/Utility/Logger/FileLc/FB_FileLc
FUNCTION_BLOCK FB_FileLc
VAR_INPUT
END_VAR
VAR_OUTPUT
END_VAR
VAR
	stFileLogClientLibInfo : T_FileLc_LibInfo;
	strInfo: Tc2_System.T_MaxString;	// additional debug Info
	bolExecute_old : BOOL;
END_VAR

(*__________________________________________________________________________________________________
¦	
¦	Vistaprint Schweiz GmbH
¦	CH - 8401 Winterthur
¦
¦	www.vistaprint.ch - info@vistaprint.ch
¦___________________________________________________________________________________________________

Function desription:
File client read out informations from BaseLog system and writes based on a config file the log entries to a file.

History:
Version		Date			Author		Comment
---------------------------------------------------------------------------------------------------
0.00.1		18.08.2014		AVME/KVO	Start history
___________________________________________________________________________________________________*)

METHOD PUBLIC M_Cyclic : UDINT
VAR_INPUT
	In_pHandle: POINTER TO T_FileLc_SysInfo; // handle for cyclic call
END_VAR
VAR
	pstSysInfo : POINTER TO T_FileLc_SysInfo;
 	pstItemDataList : POINTER TO T_FileLc_ItemData;
  	pstItemCfgList: POINTER TO T_FileLc_ItemCfg;
	stData : T_Bl_BaseStruc; // Data struct for read out
	uinReadStatus : UINT;
	ii : UINT;
	jj : UINT;
	bolWriteRecord : BOOL;
	pstrTmp : POINTER TO T_MaxString;
	strTmp:T_MaxString;
	p_Tmp_bytTmpFileBuffer : POINTER TO BYTE;
	bolKVO:BOOL;
	udiStatus : UDINT;
END_VAR
// check handle ok
IF (In_pHandle=TC3_MEMMAN.NULL) THEN
	M_Cyclic := FileLc.cERR_HANDLE;
	RETURN;
END_IF

// handle=SysInfo
pstSysInfo := In_pHandle;

// call time stamp asynchronous synchronisation
stFileLogClientLibInfo.fbTimeStamp();

// write data after a defined time to file
IF (pstSysInfo^.stFileHandler.udiWriteTimer<pstSysInfo^.stConfig.udiMaxTimeWriteToFile) THEN
	pstSysInfo^.stFileHandler.udiWriteTimer := pstSysInfo^.stFileHandler.udiWriteTimer + pstSysInfo^.udiCylceTimeMs; // add cycle time
ELSE
	pstSysInfo^.stFileHandler.udiWriteTimer := 0; // reset timer
	pstSysInfo^.stFileHandler.usiCmd := FileLc.cCMD_FLUSHBUF; // write entries to file
END_IF

// call file handler
M_Cyclic := pstSysInfo^.stFileHandler.FB_FileLc_FileHdl.M_Cyclic(In_pstSysInfo:=pstSysInfo);

(* ------------------------------------------------------------------------
Baselog buffer read out
--------------------------------------------------------------------------*)
//20 perhaps dynamic define over Level????
IF (pstSysInfo^.stItemInfo.uinActNbrOfItems>0) THEN
	FOR ii := 0 TO ((pstSysInfo^.stItemInfo.uinActNbrOfItems-1) * 20) BY 1 DO
		// Move record buffer to file buffer
		IF ((pstSysInfo^.stFileHandler.usiCmd=0) AND (pstSysInfo^.bolTmpRecordFull)) THEN
			
			// enough space in file buffer?
			IF ((pstSysInfo^.stFileHandler.udiTmpFileBufferOffset+pstSysInfo^.udiTmpRecordLen) < pstSysInfo^.stFileHandler.udiTmpFileBufferSize) THEN
			(* ----------------------------------------------------------------------------------------------------
			/* Filesize and count of records check. If the file is getting to big with the current temp buffer
			/* or the number of records in file exceed the configurated number --> Create a new file
			/* udiMaxFileSize = 0 -> no limit
			/* udiMaxEntriesInFile = 0 --> no limit
	
			/* record counter udiRecordCnt is reseted  by filhandler (new file)
			/* ----------------------------------------------------------------------------------------------------*)
	
				IF (((pstSysInfo^.stConfig.udiMaxFileSize <> 0) AND
				((pstSysInfo^.stFileHandler.udiTmpFileBufferOffset + pstSysInfo^.udiTmpRecordLen + pstSysInfo^.stFileHandler.FB_FileLc_FileHdl.ActFileSize) > pstSysInfo^.stConfig.udiMaxFileSize)) OR 
				((pstSysInfo^.stConfig.udiMaxEntriesInFile <> 0) AND (pstSysInfo^.stFileHandler.udiRecordCnt >= pstSysInfo^.stConfig.udiMaxEntriesInFile))) THEN
						
					// write to file and create new file
					pstSysInfo^.stFileHandler.usiCmd := FileLc.cCMD_FLUSHBUF_NEWFILE;
		
				ELSE 
					p_Tmp_bytTmpFileBuffer := pstSysInfo^.stFileHandler.p_bytTmpFileBuffer + pstSysInfo^.stFileHandler.udiTmpFileBufferOffset;
					
					//For Debugging
					pstrTmp := ADR(strTmp);
					MEMSET(destAddr:=pstrTmp,fillByte:=0,n:= SIZEOF(strTmp));
					MEMCPY(destAddr:=pstrTmp,srcAddr:=pstSysInfo^.p_bytTmpRecordText,n:= (SIZEOF(strTmp)-1)); // zero determining string
					
					// copy record buffer to file buffer
					memcpy(destAddr:=p_Tmp_bytTmpFileBuffer ,srcAddr:=pstSysInfo^.p_bytTmpRecordText,n:=pstSysInfo^.udiTmpRecordLen);
					
					// Filebuffer Offset increment
					pstSysInfo^.stFileHandler.udiTmpFileBufferOffset := pstSysInfo^.stFileHandler.udiTmpFileBufferOffset + pstSysInfo^.udiTmpRecordLen;
					
					// clear temp. record buffer
					pstSysInfo^.bolTmpRecordFull := FALSE;
					
					// Record Buffer ist frei -> Offset zu Null setzen
					pstSysInfo^.udiTmpRecordLen := 0;
				END_IF
			ELSE // file buffer + temp record buffer exceeds maximum
				pstSysInfo^.stFileHandler.udiWriteTimer := 0; // reset timer
				pstSysInfo^.stFileHandler.usiCmd := FileLc.cCMD_FLUSHBUF; // write file buffer to file
			END_IF
		END_IF
		
		// return if buffer still full
		IF (pstSysInfo^.bolTmpRecordFull) THEN
			RETURN;
		END_IF
			

		// reset flag
		bolWriteRecord := FALSE;
		
		// Read out from base log -> stData
		uinReadStatus := stFileLogClientLibInfo.p_fbBasLog^.M_Read(In_pHandle:=pstSysInfo^.pBaseLogHandle,In_pData:=ADR(stData)); 
		IF (uinReadStatus<>0) THEN // exit for if nothing to read
			RETURN;
		END_IF
	
		// base logging
		IF(pstSysInfo^.uinLogTyp=FileLc.cLOGTYP_BL) THEN
			//reference item list
			pstItemCfgList := pstSysInfo^.stItemInfo.p_bytItemCfgList;
			
			// on BL only use first line
			pstItemDataList := pstSysInfo^.stItemInfo.a_p_bytItemDataList[0];
			
			// must be worked on the PvId ?
			 FOR jj := 0 TO (pstSysInfo^.stItemInfo.uinActNbrOfItems-1) BY 1 DO
				 CASE (pstItemCfgList[jj].dinPvId) OF
					FileLc.cPVTYPE_BL_LOGTYP:
						M_WriteActItemIdx(In_pstItemDataList :=pstItemDataList,In_dinDataTyp:= FileLc.cVAR_TYPE_UDINT, In_pValue:=ADR(stData.udiLogType), In_udiRecIdx:=0, In_uinActItemIdx:=jj);
					FileLc.cPVTYPE_BL_CTRL_ID:
						M_WriteActItemIdx(In_pstItemDataList :=pstItemDataList,In_dinDataTyp:= FileLc.cVAR_TYPE_INT, In_pValue:=ADR(stData.intCtrlID), In_udiRecIdx:=0, In_uinActItemIdx:=jj);
					FileLc.cPVTYPE_BL_STRING1:
						M_WriteActItemIdx(In_pstItemDataList :=pstItemDataList,In_dinDataTyp:= FileLc.cVAR_TYPE_STRING, In_pValue:=ADR(stData.strText1), In_udiRecIdx:=0, In_uinActItemIdx:=jj);
					FileLc.cPVTYPE_BL_STRING2:
						M_WriteActItemIdx(In_pstItemDataList :=pstItemDataList,In_dinDataTyp:= FileLc.cVAR_TYPE_STRING, In_pValue:=ADR(stData.strText2), In_udiRecIdx:=0, In_uinActItemIdx:=jj);
					FileLc.cPVTYPE_BL_PAR1:
						M_WriteActItemIdx(In_pstItemDataList :=pstItemDataList,In_dinDataTyp:= FileLc.cVAR_TYPE_DINT, In_pValue:=ADR(stData.dinPar1), In_udiRecIdx:=0, In_uinActItemIdx:=jj);
					FileLc.cPVTYPE_BL_PAR2:
						M_WriteActItemIdx(In_pstItemDataList :=pstItemDataList,In_dinDataTyp:= FileLc.cVAR_TYPE_DINT, In_pValue:=ADR(stData.dinPar2), In_udiRecIdx:=0, In_uinActItemIdx:=jj);
					FileLc.cPVTYPE_BL_PAR3:
						M_WriteActItemIdx(In_pstItemDataList :=pstItemDataList,In_dinDataTyp:= FileLc.cVAR_TYPE_DINT, In_pValue:=ADR(stData.dinPar3), In_udiRecIdx:=0, In_uinActItemIdx:=jj);
					FileLc.cPVTYPE_BL_PAR4:
						M_WriteActItemIdx(In_pstItemDataList :=pstItemDataList,In_dinDataTyp:= FileLc.cVAR_TYPE_DINT, In_pValue:=ADR(stData.dinPar4), In_udiRecIdx:=0, In_uinActItemIdx:=jj);
							
				END_CASE
			 END_FOR
			 // general inf o add to Record list
			pstSysInfo^.stItemInfo.stItemRecordData[0].dtActDateTime := stData.dtDateTimeEntry;
			pstSysInfo^.stItemInfo.stItemRecordData[0].uinActMilli := stData.uinMs;
			
			// for BaseLog write always record 0
			M_WriteRecord(In_pstSysInfo:=pstSysInfo,In_uinItemListIdx := 0);
			
			// end of IF(pstSysInfo^.uinLogTyp=FileLc.cLOGTYP_BL) THEN
		ELSE
			(* -----------------------------------*/
		  /* Data- und PV - Logging             */
		  /* -----------------------------------*)
	
		  (* ----------------------*/
		  /* Check commandes     */
		  /* ----------------------
		  /* "cmd" in typ field *)
		  IF (stData.dinPar3 = BasLog.cVAR_TYPE_CMD_NEW_REC) THEN
	
				(* search free record - list *)
				FOR jj := 0 TO Queue.cMAX_NR_OF_TASKS BY 1 DO
				  IF ((pstSysInfo^.stItemInfo.stItemRecordData[jj].udiRecIdx = 0) OR (DINT_TO_UDINT(stData.dinPar4) = pstSysInfo^.stItemInfo.stItemRecordData[jj].udiRecIdx)) THEN
						pstSysInfo^.stItemInfo.stItemRecordData[jj].udiRecIdx := DINT_TO_UDINT(stData.dinPar4);
						pstSysInfo^.stItemInfo.stItemRecordData[jj].dtActDateTime := stData.dtDateTimeEntry;
						pstSysInfo^.stItemInfo.stItemRecordData[jj].uinActMilli := stData.uinMs;
						EXIT;
				  END_IF
			   END_FOR
		  
		  ELSIF (stData.dinPar3 = BasLog.cVAR_TYPE_CMD_END_REC) THEN
			bolWriteRecord := TRUE;
		  END_IF			
	
	
		  (* --------------------------------------------------------------*/
		  /* entry reached BaseLog message in record list */
		  /* --------------------------------------------------------------*)
		  M_PutPvIdInList(In_pstSysInfo := pstSysInfo, In_pstData := ADR(stData));
	
		  (* -----------------------------------------------------*/
		  /* write the complete record to the temporar buffer */
		  /* -----------------------------------------------------*)
		  IF (bolWriteRecord)  THEN
			FOR jj := 0 TO Queue.cMAX_NR_OF_TASKS BY 1 DO
			  (* Is the reached record index allready entried in referencelist *)
			  IF (pstSysInfo^.stItemInfo.stItemRecordData[jj].udiRecIdx = DINT_TO_UDINT(stData.dinPar4)) THEN
				M_WriteRecord(In_pstSysInfo:=pstSysInfo,In_uinItemListIdx := jj);
				EXIT;
			  END_IF
			END_FOR
		  END_IF
    END_IF // else
  END_FOR // FOR ii := 0 TO ((pstSysInfo^.stItemInfo.uinActNbrOfItems-1) * 20) BY 1 DO
END_IF 	//IF (pstSysInfo^.stItemInfo.uinActNbrOfItems>0) THEN
END_METHOD

METHOD PUBLIC M_Init : BOOL
VAR_INPUT
	In_strCfgFileName: STRING(FileLc.cFILENAME_LENGTH); // name of the config/template file
	In_strPath: STRING(FileLc.cPATH_LENGTH);  // path of the config/template file
	In_p_fbBasLog: POINTER TO FB_BasLog; // only one central FB_BasLog instance allowed per PLC!!!
	In_bolExecute : BOOL;
	In_p_uinFLcIdx : POINTER TO UINT; // actual file client id
END_VAR
VAR_OUTPUT
	Out_pHandle: POINTER TO T_FileLc_SysInfo; // handle for cyclic call	
	Out_udiStatus: UDINT; 	// 0 => successful done, <>0 => error
	Out_bolDone: BOOL;		// Done
END_VAR

VAR
	strClientName : STRING(255);
	uinFLcIdxForArr : UINT;
	udiStatus : UDINT;
	udiMask : UDINT;
	uinInitStatus : UINT;
	pQueueInfoHandle : POINTER TO POINTER TO T_Queue_Info;
	fbGETCURTASKINDEX: Tc2_System.GETCURTASKINDEX;
	udiTaskCnt : UDINT;
END_VAR
// only one client init at the same on PLC possibel!!!
IF (In_p_uinFLcIdx<>Tc3_MemMan.NULL) THEN // valid actual id reference
	IF (In_bolExecute=TRUE) THEN
		// wait until release init rom other clients...
		IF  ((stFileLogClientLibInfo.uinActClientInitActive=0) OR (stFileLogClientLibInfo.uinActClientInitActive=In_p_uinFLcIdx^)) THEN
			IF (stFileLogClientLibInfo.uinActClientInitActive=0) THEN
				stFileLogClientLibInfo.uinActClientInitActive := stFileLogClientLibInfo.uinActNbrOfFileClients + 1; // lock init of other clients!!!
				In_p_uinFLcIdx^ := stFileLogClientLibInfo.uinActClientInitActive;
				
				Out_bolDone := 0;
				Out_udiStatus := 0;
				Out_pHandle := 0;
				//reset statemachine
				(* check input parameter *)
				IF (stFileLogClientLibInfo.uinActNbrOfFileClients >= FileLc.cMAX_NBR_OF_FILECLIENTS) THEN
					Out_udiStatus := FileLc.cERR_NBR_OF_FC_EXEEDED;
					RETURN;
				END_IF
				
				IF (In_strCfgFileName='') THEN
					Out_udiStatus := FileLc.cERR_FILENAME_MISSING;
					RETURN;
				END_IF
				
				IF (In_strPath='') THEN
					Out_udiStatus := FileLc.cERR_PATH_MISSING;
					RETURN;
				END_IF
				
				IF (In_p_fbBasLog=TC3_MEMMAN.NULL) THEN
					Out_udiStatus := FileLc.cERR_NO_BASELOG;
					RETURN;
				END_IF
		
				stFileLogClientLibInfo.p_fbBasLog := In_p_fbBasLog;
				
				// actual client init
				stFileLogClientLibInfo.stSysInfo[stFileLogClientLibInfo.uinActNbrOfFileClients].stStatemachine.uinState := 1;
				stFileLogClientLibInfo.stSysInfo[stFileLogClientLibInfo.uinActNbrOfFileClients].stStatemachine.uinState_old := 0;
				stFileLogClientLibInfo.stSysInfo[stFileLogClientLibInfo.uinActNbrOfFileClients].fbFileLc_WorkOnFile(In_bolExecute:=FALSE); // reset statemachine on next positive edge!
				
				// increment client number
				stFileLogClientLibInfo.uinActNbrOfFileClients := stFileLogClientLibInfo.uinActNbrOfFileClients + 1;
				
				
			END_IF
		
			// valid client idx
			IF (In_p_uinFLcIdx^>0) THEN
				uinFLcIdxForArr := In_p_uinFLcIdx^-1; // access idx for arrays!
			
				CASE stFileLogClientLibInfo.stSysInfo[uinFLcIdxForArr].stStatemachine.uinState OF
					1:
						// check template/config file */
						stFileLogClientLibInfo.stSysInfo[uinFLcIdxForArr].fbFileLc_WorkOnFile(In_bolExecute:=TRUE,In_strPath:=In_strPath,In_strCfgFileName:=In_strCfgFileName,In_pstSysInfo := ADR(stFileLogClientLibInfo.stSysInfo[uinFLcIdxForArr]));
						IF (stFileLogClientLibInfo.stSysInfo[uinFLcIdxForArr].fbFileLc_WorkOnFile.Out_udiStatus<>0) OR (stFileLogClientLibInfo.stSysInfo[uinFLcIdxForArr].fbFileLc_WorkOnFile.Out_bolDone=1) THEN
							stFileLogClientLibInfo.stSysInfo[uinFLcIdxForArr].stStatemachine.uinState := 2;
						END_IF
						
					2:
						IF (stFileLogClientLibInfo.stSysInfo[uinFLcIdxForArr].fbFileLc_WorkOnFile.Out_udiStatus<>0) THEN // error in template/config file
							stFileLogClientLibInfo.uinActNbrOfFileClients := stFileLogClientLibInfo.uinActNbrOfFileClients - 1;
							Out_udiStatus := stFileLogClientLibInfo.stSysInfo[uinFLcIdxForArr].fbFileLc_WorkOnFile.Out_udiStatus;
							RETURN;
						END_IF
						  
						// register as client on base log system
						strClientName := BasLog.cCLIENT_NAME_PF;
						strClientName := Tc2_Standard.CONCAT(strClientName,'.fileclient');
						strClientName := Tc2_Standard.CONCAT(strClientName,UINT_TO_STRING(uinFLcIdxForArr));
						
						//LOG TYPE Maske --> PVLog Event und Cyclic 
						CASE (stFileLogClientLibInfo.stSysInfo[uinFLcIdxForArr].uinLogTyp) OF
							FileLc.cLOGTYP_DATA:
								udiMask := BasLog.cLOGTYPE_DATA;
							FileLc.cLOGTYP_PV:
								udiMask := (BasLog.cLOGTYPE_PV_EVENT OR BasLog.cLOGTYPE_PV_CYCLIC);
							FileLc.cLOGTYP_BL, FileLc.cLOGTYP_OPEN:
								udiMask := stFileLogClientLibInfo.stSysInfo[uinFLcIdxForArr].udiMask;
						END_CASE
						
						stFileLogClientLibInfo.fbTimeStamp.In_strNetId := stFileLogClientLibInfo.stSysInfo[uinFLcIdxForArr].stConfig.strLogNetId; // use system time of log target system
						stFileLogClientLibInfo.fbTimeStamp.In_t_CycleTimeRefreshTimeZone := T#0S; // cyclic check time zone settings - not needed using LocalTime_FileTime_BaseWin for log system and local time
						stFileLogClientLibInfo.p_fbBasLog^.M_ClientInit(In_strClientName:=strClientName,In_udiMask := udiMask, In_uinNrOfElement:= UDINT_TO_UINT(stFileLogClientLibInfo.stSysInfo[uinFLcIdxForArr].stConfig.udiQueueLen),In_p_fbTimeStamp:=ADR(stFileLogClientLibInfo.fbTimeStamp),In_bolUseLocalTimeStamp:=stFileLogClientLibInfo.stSysInfo[uinFLcIdxForArr].stConfig.bolUseLocalTimeStamp,Out_pHandle=>pQueueInfoHandle,Out_uinStatus=>udiStatus);
						
						IF (udiStatus<>0) THEN // check if init base log ok
							stFileLogClientLibInfo.uinActNbrOfFileClients := stFileLogClientLibInfo.uinActNbrOfFileClients - 1;
							Out_udiStatus := udiStatus;
							RETURN;
						END_IF
				
						//---------------------------------------------------------------------------------------------------------------
						// set SysInfo parameter
						stFileLogClientLibInfo.stSysInfo[uinFLcIdxForArr].pBaseLogHandle := pQueueInfoHandle;
						//DeviceName auf SysInfo Struktur ablegen
						stFileLogClientLibInfo.stSysInfo[uinFLcIdxForArr].strPathName := In_strPath;
						
						// get cycle time
						// number of tasksudiTaskCnt := TwinCAT_SystemInfoVarList._AppInfo.TaskCnt;
						fbGETCURTASKINDEX();
						udiTaskCnt := fbGETCURTASKINDEX.index;
						stFileLogClientLibInfo.stSysInfo[uinFLcIdxForArr].udiCylceTimeMs := TwinCAT_SystemInfoVarList._TaskInfo[UDINT_TO_DINT(udiTaskCnt)].CycleTime/10000; //[ms] X[100ns]/10000 -> [ms]
			
						// init filehandler
						//automatic read out infos about FUB
						udiStatus := stFileLogClientLibInfo.stSysInfo[uinFLcIdxForArr].stFileHandler.FB_FileLc_FileHdl.M_Init(In_pstSysInfo:=ADR(stFileLogClientLibInfo.stSysInfo[uinFLcIdxForArr]));
						IF (udiStatus<>0) THEN // check if init base log ok
							stFileLogClientLibInfo.uinActNbrOfFileClients := stFileLogClientLibInfo.uinActNbrOfFileClients - 1;
							Out_udiStatus := udiStatus;
							RETURN;
						END_IF
						
						// finished
						stFileLogClientLibInfo.stSysInfo[uinFLcIdxForArr].stStatemachine.uinState := 3;
					3:
						// wait for time stamp init ok (synchronize windows time, get time zone information!)
						stFileLogClientLibInfo.fbTimeStamp();
						IF (stFileLogClientLibInfo.fbTimeStamp.Out_bolInitOk) THEN
							stFileLogClientLibInfo.stSysInfo[uinFLcIdxForArr].stStatemachine.uinState := 4;
						END_IF
					4: 
						stFileLogClientLibInfo.stSysInfo[uinFLcIdxForArr].stStatemachine.usiInitDone := 1;
						Out_bolDone := TRUE; // init done
						stFileLogClientLibInfo.uinActClientInitActive := 0; // release init of other clients!!!
						// return adresse on actual SysInfo struct
						Out_pHandle := ADR(stFileLogClientLibInfo.stSysInfo[uinFLcIdxForArr]);
				END_CASE
			END_IF
		END_IF
	ELSE
		IF (stFileLogClientLibInfo.uinActClientInitActive=In_p_uinFLcIdx^) THEN // reset own flag
			stFileLogClientLibInfo.uinActClientInitActive := 0; // release init of other clients!!!
		END_IF
	END_IF
ELSE
	Out_pHandle := 0;
	Out_udiStatus := FileLc.cERR_NO_FLCIDX;
	RETURN;
END_IF
END_METHOD

METHOD PROTECTED M_PutPvIdInList : UINT
VAR_INPUT
	In_pstSysInfo: POINTER TO T_FileLc_SysInfo;
	In_pstData : POINTER TO T_Bl_BaseStruc;
END_VAR
VAR
	pstItemDataList : POINTER TO T_FileLc_ItemData;
  	pstItemCfgList: POINTER TO T_FileLc_ItemCfg;
	pstItemCfgListItem: T_FileLc_ItemCfg;
	bolItemFound : BOOL;
	uinActItemIdx : UINT;
	ii: UINT;
END_VAR
// Methode check received base log message and fill up the data to the item list
pstItemCfgList := In_pstSysInfo^.stItemInfo.p_bytItemCfgList;

bolItemFound := FALSE;

// has the id to be overworked?
FOR ii := 0 TO (In_pstSysInfo^.stItemInfo.uinActNbrOfItems-1) BY 1 DO
	pstItemCfgListItem := pstItemCfgList[ii];
	IF (pstItemCfgList[ii].dinPvId=In_pstData^.dinPar1) THEN
	 	bolItemFound := TRUE;
		uinActItemIdx := ii;
		EXIT;
	END_IF
END_FOR

// this PvId is not in list
IF (bolItemFound=FALSE) THEN
	M_PutPvIdInList := 0;
	RETURN;
END_IF

(* ---------------------------------*/
/* check reference list      */
/* and write data to the list */
/* ---------------------------------*)
FOR ii := 0 TO Queue.cMAX_NR_OF_TASKS BY 1 DO

	(* Is the received record in reference list?*)
	IF (In_pstSysInfo^.stItemInfo.stItemRecordData[ii].udiRecIdx = DINT_TO_UDINT(In_pstData^.dinPar4)) THEN
			
	  // reference to item list
	  pstItemDataList := In_pstSysInfo^.stItemInfo.a_p_bytItemDataList[ii];
	
	  (* write data to item list *)
	  IF (In_pstData^.dinPar3 = FileLc.cVAR_TYPE_STRING) THEN// data definition
		M_WriteActItemIdx(In_pstItemDataList :=pstItemDataList,In_dinDataTyp:= FileLc.cVAR_TYPE_STRING, In_pValue:=ADR(In_pstData^.strText2), In_udiRecIdx:=DINT_TO_UDINT(In_pstData^.dinPar4), In_uinActItemIdx:=uinActItemIdx);
	  ELSE
		M_WriteActItemIdx(In_pstItemDataList:=pstItemDataList, In_dinDataTyp := In_pstData^.dinPar3, In_pValue := ADR(In_pstData^.dinPar2),In_udiRecIdx := DINT_TO_UDINT(In_pstData^.dinPar4), In_uinActItemIdx := uinActItemIdx);
	  END_IF
	  EXIT;
	END_IF
END_FOR		

M_PutPvIdInList := 0;
RETURN;
END_METHOD

METHOD PROTECTED M_ReleaseBuffer : UINT

VAR_INPUT
	In_pReleaseBuffer : POINTER TO BYTE;
END_VAR
//delocate  allocated buffer with __NEW
__DELETE(In_pReleaseBuffer);
RETURN; // delete buffer with dynamic size...
END_METHOD

METHOD PROTECTED M_WriteActItemIdx : UINT
VAR_INPUT
	In_pstItemDataList : POINTER TO T_FileLc_ItemData;
	In_dinDataTyp: DINT;
	In_pValue: POINTER TO BYTE;
	In_udiRecIdx : UDINT;
	In_uinActItemIdx : UINT;
END_VAR

VAR
	strTmp : T_MaxString;
	pString : POINTER TO STRING(255);
	pBool : POINTER TO BOOL;
	pSint : POINTER TO SINT;
	pInt : POINTER TO INT;
	pDint : POINTER TO DINT;
	pUsint : POINTER TO USINT;
	pUint : POINTER TO UINT;
	pUdint : POINTER TO UDINT;
	pReal : POINTER TO REAL;
	pLreal : POINTER TO LREAL;
	stItemDataListItem : T_FileLc_ItemData;
END_VAR
// write value in ItemList based on datatyp
IF (In_pValue<>TC3_MEMMAN.NULL) THEN
	 CASE In_dinDataTyp OF
		FileLc.cVAR_TYPE_SINT:
			pSint := In_pValue;
			strTmp := SINT_TO_STRING(pSint^);	
		FileLc.cVAR_TYPE_INT:
			pInt := In_pValue;
			strTmp := INT_TO_STRING(pInt^);
		FileLc.cVAR_TYPE_DINT:
			pDint := In_pValue;
			strTmp := DINT_TO_STRING(pDint^);
		FileLc.cVAR_TYPE_BOOL:
			pBool := In_pValue;
			strTmp := BOOL_TO_STRING(pBool^);	
		FileLc.cVAR_TYPE_USINT:
			pUsint := In_pValue;
			strTmp := USINT_TO_STRING(pUsint^);
		FileLc.cVAR_TYPE_UINT:
			pUint := In_pValue;
			strTmp := UINT_TO_STRING(pUint^);
		FileLc.cVAR_TYPE_UDINT:
			pUdint := In_pValue;
			strTmp := UDINT_TO_STRING(pUdint^);
		FileLc.cVAR_TYPE_REAL:
			pReal := In_pValue;
			strTmp := REAL_TO_STRING(pReal^);
		FileLc.cVAR_TYPE_LREAL:
			pLreal := In_pValue;
			strTmp := LREAL_TO_STRING(pLreal^);
		FileLc.cVAR_TYPE_STRING:
			pString := In_pValue;
			strTmp := pString^;
		ELSE
			strTmp := 'unknown type';
	END_CASE
	
	IF (INT_TO_UINT(LEN(strTmp)) >=  FileLc.cMAX_ITEM_CHAR) THEN
		In_pstItemDataList[In_uinActItemIdx].strValue:= 'value too long';
	ELSE
		MEMSET(destAddr := ADR(In_pstItemDataList[In_uinActItemIdx].strValue),0,SIZEOF(In_pstItemDataList[In_uinActItemIdx].strValue)); // string ends wit 0!
		MEMCPY(destAddr := ADR(In_pstItemDataList[In_uinActItemIdx].strValue),srcAddr:=ADR(strTmp),SIZEOF(strTmp));
	END_IF
END_IF
// entry record index
In_pstItemDataList[In_uinActItemIdx].udiRecIdx := In_udiRecIdx;
stItemDataListItem := In_pstItemDataList[In_uinActItemIdx]; // for Debugging
END_METHOD

METHOD PROTECTED M_WriteRecord : UINT
VAR_INPUT
	In_pstSysInfo: POINTER TO T_FileLc_SysInfo;
	In_uinItemListIdx : UINT;
END_VAR
VAR
 	pstItemDataList : POINTER TO T_FileLc_ItemData;
  	pstItemCfgList: POINTER TO T_FileLc_ItemCfg;
	pstItemCfgListItem: T_FileLc_ItemCfg;
	pstItemDataListItem : T_FileLc_ItemData;
	pstRecordData : POINTER TO T_FileLc_RecordData;
	ii : UINT;
	bolRecordValid : BOOL;
	udiOffset : UDINT;
	udiTmpLen : UDINT;
	strTemp : STRING(30);
	SystemTimeStruct  :TIMESTRUCT;
END_VAR
pstItemDataList := In_pstSysInfo^.stItemInfo.a_p_bytItemDataList[In_uinItemListIdx];
pstItemCfgList := In_pstSysInfo^.stItemInfo.p_bytItemCfgList;
pstRecordData := ADR(In_pstSysInfo^.stItemInfo.stItemRecordData[In_uinItemListIdx]);

// copy PRE - Text
udiOffset := 0;
udiTmpLen := INT_TO_UDINT(LEN(In_pstSysInfo^.stItemInfo.strPreItemText));
MEMCPY(destAddr := (In_pstSysInfo^.p_bytTmpRecordText+udiOffset),srcAddr :=ADR(In_pstSysInfo^.stItemInfo.strPreItemText) , n := udiTmpLen);
udiOffset := udiOffset + udiTmpLen;

// check filled data
bolRecordValid := FALSE;
//at least one item has to be added before
FOR ii := 0 TO (In_pstSysInfo^.stItemInfo.uinActNbrOfItems-1) BY 1 DO
	pstItemCfgListItem := pstItemCfgList[ii];
	pstItemDataListItem := pstItemDataList[ii];
	IF ((pstItemCfgListItem.dinPvId>=0) AND (pstItemDataListItem.udiRecIdx=pstRecordData^.udiRecIdx)) THEN
	 	bolRecordValid := TRUE;
		 EXIT;
	END_IF
END_FOR

// record has no valid data
IF ((bolRecordValid=FALSE) AND (In_pstSysInfo^.uinLogTyp<>FileLc.cLOGTYP_BL)) THEN
	// clear record data
	pstRecordData^.udiRecIdx :=0;
	pstRecordData^.dtActDateTime := REAL_TO_DT(0.0);
	pstRecordData^.uinActMilli :=0;
	
	// reset record buffer
	In_pstSysInfo^.udiTmpRecordLen := 0;
	In_pstSysInfo^.bolTmpRecordFull := FALSE;
	RETURN;
END_IF

// collect data
FOR ii := 0 TO (In_pstSysInfo^.stItemInfo.uinActNbrOfItems-1) BY 1 DO
	//for debugging
	pstItemCfgListItem := pstItemCfgList[ii];
	pstItemDataListItem := pstItemDataList[ii];
	
	IF (pstItemCfgListItem.dinPvId<0) THEN
	 	CASE (pstItemCfgListItem.dinPvId) OF
			FileLc.cPVTYPE_UNIX_DATE_TIME_STR:
				// time and date as string
				pstItemDataListItem.strValue := DT_TO_STRING(pstRecordData^.dtActDateTime);
			
			FileLc.cPVTYPE_UNIX_DATE_TIME:
				// time and date as  s since 1.1.1970 11:00
				pstItemDataListItem.strValue := DWORD_TO_STRING(DT_TO_DWORD(pstRecordData^.dtActDateTime));
			
			FileLc.cPVTYPE_EXCEL_DATE_TIME:
				// time and date as REAL
				pstItemDataListItem.strValue := LREAL_TO_STRING(DT_TO_LREAL(pstRecordData^.dtActDateTime));
				(*needed ?? if (pdstRecordData->dtActDateTime > 0) {
						tmpDouble = (double)(pdstRecordData->dtActDateTime / 86400.0) + 25569.0;
						tmpUdint = (double)tmpDouble;  /*Ganzzahl bilden/
						tmpDouble = (tmpDouble - tmpUdint); /*Nachkommastellen/
						itoa(tmpUdint, (unsigned long)&pdstItemDataList[i].strValue);
						strcat((void)&pdstItemDataList[i].strValue, ".");

						// Nachkommaanteil mit 10 hoch n multipizieren
						tmpUdint = tmpDouble * tmpPrecision;
	
						// Integer to ACSI Wandlung mit Vornullen!
						tmpPrecision = tmpPrecision / 10;
						n=0;
						while (tmpPrecision > 1) {
							tmpString[n] = (tmpUdint / tmpPrecision) + 0x30;  // Character Wandlung
							tmpUdint = tmpUdint % tmpPrecision;
							tmpPrecision = tmpPrecision / 10;
							n++;
						}
						tmpString[n]=0;
						strcat((void)&pdstItemDataList[i].strValue, (void)&tmpString);
						ulSize = strlen(pdstItemDataList[i].strValue);
					}*)
			FileLc.cPVTYPE_DATE_SLASH_TIME_COLON: 
				//english date format 2014/09/23 07:10:24
				SystemTimeStruct := DT_TO_SYSTEMTIME(pstRecordData^.dtActDateTime);
				pstItemDataListItem.strValue := DWORD_TO_STRING(SystemTimeStruct.wYear);
				pstItemDataListItem.strValue := CONCAT(STR1:=pstItemDataListItem.strValue,STR2:='/');
				IF (SystemTimeStruct.wMonth<10) THEN
					pstItemDataListItem.strValue := CONCAT(pstItemDataListItem.strValue , '0');
				END_IF
				pstItemDataListItem.strValue := CONCAT(STR1:=pstItemDataListItem.strValue,STR2:=DWORD_TO_STRING(SystemTimeStruct.wMonth));
				pstItemDataListItem.strValue := CONCAT(STR1:=pstItemDataListItem.strValue,STR2:='/');
				IF (SystemTimeStruct.wDay<10) THEN
					pstItemDataListItem.strValue := CONCAT(pstItemDataListItem.strValue , '0');
				END_IF
				pstItemDataListItem.strValue := CONCAT(STR1:=pstItemDataListItem.strValue,STR2:=DWORD_TO_STRING(SystemTimeStruct.wDay));
				pstItemDataListItem.strValue := CONCAT(STR1:=pstItemDataListItem.strValue,STR2:=' ');
				IF (SystemTimeStruct.wHour<10) THEN
					pstItemDataListItem.strValue := CONCAT(pstItemDataListItem.strValue , '0');
				END_IF
				pstItemDataListItem.strValue := CONCAT(STR1:=pstItemDataListItem.strValue,STR2:=DWORD_TO_STRING(SystemTimeStruct.wHour));
				pstItemDataListItem.strValue := CONCAT(STR1:=pstItemDataListItem.strValue,STR2:=':');
				IF (SystemTimeStruct.wMinute<10) THEN
					pstItemDataListItem.strValue := CONCAT(pstItemDataListItem.strValue , '0');
				END_IF
				pstItemDataListItem.strValue := CONCAT(STR1:=pstItemDataListItem.strValue,STR2:=DWORD_TO_STRING(SystemTimeStruct.wMinute));
				pstItemDataListItem.strValue := CONCAT(STR1:=pstItemDataListItem.strValue,STR2:=':');
				IF (SystemTimeStruct.wSecond<10) THEN
					pstItemDataListItem.strValue := CONCAT(pstItemDataListItem.strValue , '0');
				END_IF
				pstItemDataListItem.strValue := CONCAT(STR1:=pstItemDataListItem.strValue,STR2:=DWORD_TO_STRING(SystemTimeStruct.wSecond));
			FileLc.cPVTYPE_TIME_MILLI:
				IF (pstRecordData^.uinActMilli<100) THEN
					IF (pstRecordData^.uinActMilli<10) THEN
						pstItemDataListItem.strValue := '00';
					ELSE
						pstItemDataListItem.strValue := '0';
					END_IF
				ELSE
					pstItemDataListItem.strValue := '';
				END_IF
				pstItemDataListItem.strValue := CONCAT(STR1:=pstItemDataListItem.strValue,STR2:=UINT_TO_STRING(pstRecordData^.uinActMilli));
		END_CASE
	END_IF
	
	
	(* ----------------------------------*/ 
	/* Write data to temp buffer */
	/* ----------------------------------*/ 
	/* PV value *)		
	IF ((pstItemDataListItem.udiRecIdx = pstRecordData^.udiRecIdx) OR (pstItemCfgListItem.dinPvId < 0)) THEN
		udiTmpLen := INT_TO_UDINT(LEN(pstItemDataListItem.strValue));
		MEMCPY(destAddr := (In_pstSysInfo^.p_bytTmpRecordText+udiOffset),srcAddr :=ADR(pstItemDataListItem.strValue) , n := udiTmpLen);
	ELSE 
		strTemp := 'no val.';
		udiTmpLen := INT_TO_UDINT(LEN(strTemp)); 
		MEMCPY(destAddr := (In_pstSysInfo^.p_bytTmpRecordText+udiOffset),srcAddr :=ADR(strTemp) , n := udiTmpLen);	
	END_IF
	udiOffset := udiOffset + udiTmpLen;
	
	IF (ii>0) AND (ii=In_pstSysInfo^.stItemInfo.uinActNbrOfItems-1) AND (udiTmpLen=0) THEN // last text empty...
		// remove last post text...
		udiTmpLen := INT_TO_UDINT(LEN(pstItemCfgList[ii-1].strPostText));
		IF (udiOffset>udiTmpLen) THEN
			MEMSET(destAddr := (In_pstSysInfo^.p_bytTmpRecordText+udiOffset-udiTmpLen),fillByte :=0 , n := udiTmpLen);
			udiOffset := udiOffset - udiTmpLen;
		END_IF
	END_IF
	
	(* Post Text *)	
	udiTmpLen := INT_TO_UDINT(LEN(pstItemCfgListItem.strPostText));
	MEMCPY(destAddr := (In_pstSysInfo^.p_bytTmpRecordText+udiOffset),srcAddr :=ADR(pstItemCfgListItem.strPostText) , n := udiTmpLen);
	udiOffset := udiOffset + udiTmpLen;

END_FOR(*for (i = 0; i < pdstSysInfo->dstItemInfo.uinActNbrOfItems; i++) *)


(* carriage return on end of record *)
udiTmpLen := SIZEOF(FileLc.cEOL);
MEMCPY(destAddr := (In_pstSysInfo^.p_bytTmpRecordText+udiOffset),srcAddr :=ADR(FileLc.cEOL) , n := udiTmpLen);
udiOffset := udiOffset + udiTmpLen;

// clear record data
pstRecordData^.udiRecIdx :=0;
pstRecordData^.dtActDateTime :=REAL_TO_DT(0.0);
pstRecordData^.uinActMilli :=0;

// mark record buffer as full
In_pstSysInfo^.udiTmpRecordLen := udiOffset;
In_pstSysInfo^.bolTmpRecordFull := TRUE;

(*--------------------------------*/
/* count file entries */
/*--------------------------------*)
In_pstSysInfo^.stFileHandler.udiRecordCnt := In_pstSysInfo^.stFileHandler.udiRecordCnt + 1;
END_METHOD

END_FUNCTION_BLOCK

// POUs/Utility/Logger/FileLc/FB_FileLc_FileHdl
FUNCTION_BLOCK FB_FileLc_FileHdl
VAR_INPUT
END_VAR
VAR_OUTPUT
END_VAR
VAR
	fbFileHdl : FB_FileHdl;
	bol_fpNewFileEvent : BOOL;
END_VAR

PROPERTY PUBLIC ActFileSize : UDINT
GET
ActFileSize := fbFileHdl.ActFileSize;
END_GET
END_PROPERTY

METHOD PUBLIC M_Cyclic : UDINT
VAR_INPUT
	In_pstSysInfo: POINTER TO T_FileLc_SysInfo;
END_VAR

VAR

END_VAR
VAR CONSTANT
	// specific steps definitions
	cStep_Wait4Job: UINT := 500;
	cStep_WriteFileBuf: UINT := 501;
	cStep_WriteFooter: UINT := 502;
	cStep_CreateNew: UINT := 503;
	cStep_WriteHeader: UINT := 504;
END_VAR
fbFileHdl();

CASE In_pstSysInfo^.stFileHandler.uinState OF
	0:	In_pstSysInfo^.stFileHandler.uinState := cStep_Wait4Job;
	
	// ready for new job
	cStep_Wait4Job:
		IF (In_pstSysInfo^.stFileHandler.uinState<>In_pstSysInfo^.stFileHandler.uinState_old) THEN
			In_pstSysInfo^.stFileHandler.strInfo := 'I: cStep_Wait4Job';
			
			In_pstSysInfo^.stFileHandler.uinState_old := In_pstSysInfo^.stFileHandler.uinState;
		END_IF
		
		// file handler ready for new commands
		IF (fbFileHdl.Out_bolBusy=FALSE) THEN
			// create new file after startup
			IF ((In_pstSysInfo^.stConfig.uinNewFileOnRestart=1) AND (In_pstSysInfo^.stFileHandler.usiInitDone=0)) THEN
				In_pstSysInfo^.stFileHandler.usiCmdNewFile := 1; 
			END_IF
			
			// mark for restart detection
			In_pstSysInfo^.stFileHandler.usiInitDone := 1;	

			// event from filehandler nwe file created!!!
			IF (fbFileHdl.Out_bolNewFileCreated) THEN
				IF (bol_fpNewFileEvent=FALSE) THEN // detect positive edge on signal!!
					bol_fpNewFileEvent := TRUE;
					In_pstSysInfo^.stFileHandler.uinState := cStep_WriteHeader;
				END_IF
			ELSE
				bol_fpNewFileEvent := FALSE;
			END_IF
			
			// finish file
			IF (In_pstSysInfo^.stFileHandler.usiCmdNewFile=1) THEN
				In_pstSysInfo^.stFileHandler.usiCmd := FileLc.cCMD_FLUSHBUF_NEWFILE;
				In_pstSysInfo^.stFileHandler.usiCmdNewFile :=0;
			END_IF
			
			// temp file buffer write to file
			IF ((In_pstSysInfo^.stFileHandler.usiCmd=FileLc.cCMD_FLUSHBUF_NEWFILE) OR (In_pstSysInfo^.stFileHandler.usiCmd=FileLc.cCMD_FLUSHBUF)) THEN
				In_pstSysInfo^.stFileHandler.uinState :=cStep_WriteFileBuf;
				
			END_IF
		END_IF
	
	// write file buffer to file
	cStep_WriteFileBuf:
		// entry action
		IF (In_pstSysInfo^.stFileHandler.uinState<>In_pstSysInfo^.stFileHandler.uinState_old) THEN
			In_pstSysInfo^.stFileHandler.strInfo := 'I: cStep_WriteFileBuf';
			
			fbFileHdl.M_Cmd_WriteBuffer(In_p_bytWriteBuff:=In_pstSysInfo^.stFileHandler.p_bytTmpFileBuffer,In_udiWriteLen:=In_pstSysInfo^.stFileHandler.udiTmpFileBufferOffset);
			fbFileHdl(); // first call -> set busy flag = TRUE
			
			In_pstSysInfo^.stFileHandler.uinState_old := In_pstSysInfo^.stFileHandler.uinState;
		END_IF
		
		fbFileHdl(); // first call -> set busy flag = TRUE
		
		// always action
		IF (fbFileHdl.Out_bolBusy=FALSE) THEN
			IF (fbFileHdl.Out_udiErrId<>0) THEN
				In_pstSysInfo^.stFileHandler.usiCmd := 0;
				In_pstSysInfo^.stFileHandler.uinState :=cStep_WriteFooter;
			ELSIF (In_pstSysInfo^.stFileHandler.usiCmd=FileLc.cCMD_FLUSHBUF) THEN
				// reset file buffer and add offset
				In_pstSysInfo^.stFileHandler.udiTmpFileBufferOffset := 0;
				In_pstSysInfo^.stFileHandler.usiCmd := 0;
				In_pstSysInfo^.stFileHandler.uinState :=cStep_Wait4Job;
			ELSIF (In_pstSysInfo^.stFileHandler.usiCmd=FileLc.cCMD_FLUSHBUF_NEWFILE) THEN
				// reset file buffer and add offset
				In_pstSysInfo^.stFileHandler.udiTmpFileBufferOffset := 0;
				In_pstSysInfo^.stFileHandler.uinState :=cStep_WriteFooter;
			END_IF
		END_IF
		
	// write footer to file
	cStep_WriteFooter:
		// entry action
		IF (In_pstSysInfo^.stFileHandler.uinState<>In_pstSysInfo^.stFileHandler.uinState_old) THEN
			In_pstSysInfo^.stFileHandler.strInfo := 'I: cStep_WriteFooter';
			
			fbFileHdl.M_Cmd_WriteBuffer(In_p_bytWriteBuff:=In_pstSysInfo^.p_bytFooterText,In_udiWriteLen:=In_pstSysInfo^.udiFooterTextLen);
			fbFileHdl(); // first call -> set busy flag = TRUE
			
			In_pstSysInfo^.stFileHandler.uinState_old := In_pstSysInfo^.stFileHandler.uinState;
		END_IF
		
		fbFileHdl(); // first call -> set busy flag = TRUE
		
		// always action
		IF (fbFileHdl.Out_bolBusy=FALSE) THEN
			IF (fbFileHdl.Out_udiErrId<>0) THEN
				In_pstSysInfo^.stFileHandler.uinState :=cStep_CreateNew;
			ELSE
				In_pstSysInfo^.stFileHandler.uinState :=cStep_CreateNew;
			END_IF
		END_IF
		
	// create new file
	cStep_CreateNew:
		// entry action
		IF (In_pstSysInfo^.stFileHandler.uinState<>In_pstSysInfo^.stFileHandler.uinState_old) THEN
			In_pstSysInfo^.stFileHandler.strInfo := 'I: cStep_CreateNew';
			
			fbFileHdl.M_Cmd_NewFile();
			fbFileHdl(); // first call -> set busy flag = TRUE
			
			In_pstSysInfo^.stFileHandler.uinState_old := In_pstSysInfo^.stFileHandler.uinState;
		END_IF
		
		fbFileHdl(); // first call -> set busy flag = TRUE
		
		// always action
		IF (fbFileHdl.Out_bolBusy=FALSE) THEN
			In_pstSysInfo^.stFileHandler.uinState := cStep_WriteHeader;
		END_IF
		
	// create new file
	cStep_WriteHeader:
		// entry action
		IF (In_pstSysInfo^.stFileHandler.uinState<>In_pstSysInfo^.stFileHandler.uinState_old) THEN
			In_pstSysInfo^.stFileHandler.strInfo := 'I: cStep_WriteHeader';
			
			fbFileHdl.M_Cmd_WriteBuffer(In_p_bytWriteBuff:=In_pstSysInfo^.p_bytHeaderText,In_udiWriteLen:=In_pstSysInfo^.udiHeaderTextLen);
			fbFileHdl(); // first call -> set busy flag = TRUE
			
			In_pstSysInfo^.stFileHandler.uinState_old := In_pstSysInfo^.stFileHandler.uinState;
		END_IF
		
		fbFileHdl(); // first call -> set busy flag = TRUE
		
		// always action
		IF (fbFileHdl.Out_bolBusy=FALSE) THEN
			In_pstSysInfo^.stFileHandler.usiCmd := 0;
			In_pstSysInfo^.stFileHandler.uinState := cStep_Wait4Job;
		END_IF
END_CASE

fbFileHdl();

M_Cyclic := fbFileHdl.Out_udiErrId; // error number feedback, reset with next job
END_METHOD

METHOD PUBLIC M_Init : UDINT
VAR_INPUT
	In_pstSysInfo: POINTER TO T_FileLc_SysInfo;
END_VAR
// max file size set higher than defined because of writing footer before create new file -> FileLc manages max file size!!!
fbFileHdl.M_Init(In_strNetId := In_pstSysInfo^.stConfig.strLogNetId ,IN_strPath:= In_pstSysInfo^.stConfig.strLogPath,IN_strFileName:=In_pstSysInfo^.stConfig.strLogFileNamePraeFix,IN_strFileExt:=In_pstSysInfo^.stConfig.strLogFileNameExt,IN_uinMaxNrOfFilesInFolder:=In_pstSysInfo^.stConfig.uinMaxNbrOfLogFiles,IN_lreMaxFileSize:=(UDINT_TO_REAL(In_pstSysInfo^.stConfig.udiMaxFileSize)*1.2),IN_timFileSupervisionPeriod:=UDINT_TO_TIME(In_pstSysInfo^.stConfig.udiTimeCheckMaxFileNr));
M_Init := fbFileHdl.Out_udiErrId;
END_METHOD

END_FUNCTION_BLOCK

// POUs/Utility/Logger/FileLc/FB_FileLc_WorkOnFile
FUNCTION_BLOCK FB_FileLc_WorkOnFile
VAR_INPUT
	In_strCfgFileName: STRING(FileLc.cFILENAME_LENGTH); // name of the config/template file (not implemented yet)
	In_strPath: STRING(FileLc.cPATH_LENGTH); 
	In_pstSysInfo : POINTER TO T_FileLc_SysInfo;
	In_bolExecute : BOOL;
END_VAR
VAR_OUTPUT
	Out_udiStatus: UDINT;			// Rückgabewert 0:ok
	Out_bolDone: BOOL;			// Done
END_VAR
VAR
	fbFileOpen : FB_FileOpen;
	fbFileRead : FB_FileRead;
	fbFileClose : FB_FileClose;
	fbFileSeek : FB_FileSeek;
	udiWaitFileOpenCycles : UDINT;
	udiWaitFileReadCycles : UDINT;
	uinFileSize: UINT := 1000; // nr of Bytes to read whole config file
	p_bytTemplateBegin : POINTER TO BYTE;
	p_bytTemplateEnd : POINTER TO BYTE;
	p_bytConfigBegin : POINTER TO BYTE;
	p_bytConfigEnd : POINTER TO BYTE;
	p_bytHeaderBegin : POINTER TO BYTE;
	p_bytHeaderEnd : POINTER TO BYTE;
	p_bytFooterBegin : POINTER TO BYTE;
	p_bytFooterEnd : POINTER TO BYTE;
	p_bytRecordBegin : POINTER TO BYTE;
	p_bytRecordEnd : POINTER TO BYTE;
	p_bytTmpDestAdr : POINTER TO BYTE;
	p_bytTmpSrcAdr : POINTER TO BYTE;
	p_bytRowBegin : POINTER TO BYTE;
	p_bytRowEnd : POINTER TO BYTE;
	p_bytItemBegin : POINTER TO BYTE;
	p_bytItemEnd : POINTER TO BYTE;
	p_bytLastPos : POINTER TO BYTE;
	p_bytConfigValBegin : POINTER TO BYTE;
	p_bytConfigValEnd : POINTER TO BYTE;
	uinTmpLen : UINT;
	uinItemCount : UINT;
	ii : USINT;
	p_stItemCfgList : POINTER TO T_FileLc_ItemCfg;
	udiTmpLen : UDINT;
	strTmp : T_MaxString;
	udiWaitFileCloseCycles : UDINT := 0;
	bolBufferNotOk : BOOL;
	udiFileConfigLen : UDINT;
	pstrTmp : POINTER TO T_MaxString;
	strTmpTest:T_MaxString;
	stStatemachine : T_FileLc_Statemachine;
	strInfo :T_MaxString;
	bolExecute_old : BOOL;
	bolTmp : BOOL;
	pDelReadPointer : POINTER TO BYTE;
END_VAR

IF (In_bolExecute=TRUE) THEN
	IF (bolExecute_old=FALSE) THEN
		//reset statemachine
		stStatemachine.uinState :=0;
		stStatemachine.uinState_old := 255;
		Out_bolDone := 0;
		Out_udiStatus := 0;
	END_IF
	;
	
	CASE stStatemachine.uinState OF
		0: 
			IF (In_strCfgFileName<>'') THEN
				Out_bolDone := FALSE;
				strInfo := '';
				Out_udiStatus := 0;
				pstrTmp := ADR(strTmpTest);
				stStatemachine.uinState := stStatemachine.uinState  + 1;
			END_IF
		1: 
			// Entry action
			IF (stStatemachine.uinState_old <> stStatemachine.uinState) THEN
				//---------------------------------------------------------
				// File parser and check settings/configs
				//---------------------------------------------------------
				
				//*********************************************************
				// file open
				fbFileOpen.sNetId := ''; // only local access
				fbFileOpen.sPathName := CONCAT(STR1:=In_strPath,STR2:=In_strCfgFileName);
				fbFileOpen.nMode := Tc2_System.FOPEN_MODEREAD OR FOPEN_MODETEXT;      // Opens for reading in text format
				fbFileOpen.ePath := PATH_GENERIC;
				fbFileOpen.tTimeout := T#30S;
				fbFileOpen(bExecute:= FALSE);
				fbFileOpen(bExecute:= TRUE);
				
				// wait until fail isopened
				udiWaitFileOpenCycles := 0;
				 stStatemachine.uinState_old := stStatemachine.uinState;
			END_IF
			
			fbFileOpen(bExecute:= TRUE);
			
			IF ((fbFileOpen.bError=FALSE) AND ((fbFileOpen.bBusy) OR (fbFileOpen.hFile=0))) THEN
				udiWaitFileOpenCycles := udiWaitFileOpenCycles + 1;	
			ELSE
				IF (fbFileOpen.bError=TRUE) THEN
					// file not found
					IF (fbFileOpen.nErrId=16#70C) THEN
						strInfo := CONCAT(STR1:='template/config file: not found: ',STR2:= In_strPath); 
						strInfo := CONCAT(STR1:=strInfo,STR2:= In_strCfgFileName); 
						Out_udiStatus := fbFileOpen.nErrId;
						RETURN;
					ELSE 
						strInfo := CONCAT(STR1:='template/config file: no more free file handles / unknown or invalid nMode or ePath parameter: ',STR2:= In_strPath); 
						strInfo := CONCAT(STR1:=strInfo,STR2:= In_strCfgFileName); 
						Out_udiStatus := fbFileOpen.nErrId;
						RETURN;
					END_IF
				ELSE
					stStatemachine.uinState := 3;
				END_IF
			END_IF
		
		3:	// read config file in temp buffer allocate buffer
			// Entry action
			IF (stStatemachine.uinState_old <> stStatemachine.uinState) THEN
				//*********************************************************
				// read template file
				fbFileRead.sNetId:=''; // local file access
				fbFileRead.hFile:=fbFileOpen.hFile;
				fbFileRead.tTimeout:=T#3S;
				// create buffer
				fbFileRead.pReadBuff := M_AllocMEM(uinFileSize);
				pDelReadPointer := fbFileRead.pReadBuff; // pointer for release
				fbFileRead.cbReadLen := uinFileSize;
				
				IF (fbFileRead.pReadBuff=TC3_MEMMAN.NULL) THEN
					strInfo := CONCAT(STR1:='template/config file: alloc file buffer invalid: ',STR2:= In_strPath);
					strInfo := CONCAT(STR1:=strInfo,STR2:= In_strCfgFileName);
					Out_udiStatus := FileLc.cERR_ALLOC_BUFFER_FILE_CONFIG;
					RETURN;
				END_IF
				
				//valid buffer allocated
				fbFileRead(bExecute:=FALSE);
				fbFileRead(bExecute:=TRUE);
				udiWaitFileReadCycles := 0;
					
				 stStatemachine.uinState_old := stStatemachine.uinState;
			END_IF
			
			fbFileRead();	
			
			// read file binary
			IF (fbFileRead.bBusy) THEN
				udiWaitFileReadCycles := udiWaitFileReadCycles + 1;
			ELSE
				
			//test variabel
		MEMSET(destAddr:=pstrTmp,fillByte:=0,n:= SIZEOF(strTmp));
		MEMCPY(destAddr:=pstrTmp,srcAddr:=fbFileRead.pReadBuff,n:= (SIZEOF(strTmp)-1)); // zero determining string
		
				IF (fbFileRead.bError=FALSE) THEN
					IF (fbFileRead.cbRead<UINT_TO_UDINT(uinFileSize)) THEN // enough memory for whole cfg file allocated
						// allocated buffer is ok
						udiFileConfigLen := fbFileRead.cbRead; // file len read
						stStatemachine.uinState := stStatemachine.uinState  + 1;
					ELSE
						// buffer size to small! 
						
						// reset file read pointer
						fbFileSeek.sNetId:=''; // local file access
						fbFileSeek.hFile:=fbFileOpen.hFile;
						fbFileSeek.eOrigin:=E_SeekOrigin.SEEK_SET; // start pos at beginning of file
						fbFileSeek.tTimeout:=T#3S;
						fbFileSeek.nSeekPos := 0; // at beginn of file
						fbFileSeek(bExecute:=FALSE);
						fbFileSeek(bExecute:=TRUE);
						WHILE (fbFileSeek.bBusy) DO
							udiWaitFileReadCycles := udiWaitFileReadCycles + 1;
							fbFileSeek(bExecute:=TRUE);
						END_WHILE
						
						//release old buffer
						__DELETE(pDelReadPointer);

						uinFileSize := LREAL_TO_UINT(UINT_TO_LREAL(uinFileSize) * 1.5); // create bigger buffer for next try
						
						stStatemachine.uinState_old := 0; // entry action alloc new buffer
					END_IF
					
				ELSE
					// error read file
					strInfo := CONCAT(STR1:='template/config file: error reading file: ',STR2:= In_strPath);
					strInfo := CONCAT(STR1:=strInfo,STR2:= In_strCfgFileName);
					Out_udiStatus := fbFileRead.nErrId;
					RETURN;
				END_IF;
			END_IF
				
			
			
		4:
			//*********************************************************	
			// parse template file
			// <TEMPLATE>pBuffer
			p_bytTemplateBegin := strstr(In_pStr:=fbFileRead.pReadBuff,In_pStrSearch:=ADR(FileLc.cTAG_TEMPLATE_B),In_bolAddStrSearchLen:= TRUE);
			p_bytTemplateEnd := strstr(In_pStr:=fbFileRead.pReadBuff,In_pStrSearch:=ADR(FileLc.cTAG_TEMPLATE_E),In_bolAddStrSearchLen:= FALSE);
			IF ((p_bytTemplateBegin=TC3_MEMMAN.NULL) OR (p_bytTemplateEnd=TC3_MEMMAN.NULL) OR (p_bytTemplateBegin>p_bytTemplateEnd)) THEN
				strInfo := CONCAT(STR1:='template/config file: parse error: ',STR2:= FileLc.cTAG_TEMPLATE_B);
				Out_udiStatus := FileLc.cERR_TEMPLATE_TAG;
				RETURN;
			END_IF
			
			// <CONFIG>
			p_bytConfigBegin := strstr(In_pStr:=fbFileRead.pReadBuff,In_pStrSearch:=ADR(FileLc.cTAG_CONFIG_B),In_bolAddStrSearchLen:= TRUE);
			p_bytConfigEnd := strstr(In_pStr:=fbFileRead.pReadBuff,In_pStrSearch:=ADR(FileLc.cTAG_CONFIG_E),In_bolAddStrSearchLen:= FALSE);
		
			IF ((p_bytConfigBegin=TC3_MEMMAN.NULL) OR (p_bytConfigEnd=TC3_MEMMAN.NULL) OR (p_bytConfigBegin>p_bytConfigEnd)) THEN
				strInfo := CONCAT(STR1:='template/config file: parse error: ',STR2:= FileLc.cTAG_CONFIG_B);
				Out_udiStatus := FileLc.cERR_CONFIG_TAG;
				RETURN;
			END_IF
			
			// <HEADER>
			p_bytHeaderBegin := strstr(In_pStr:=fbFileRead.pReadBuff,In_pStrSearch:=ADR(FileLc.cTAG_HEADER_B),In_bolAddStrSearchLen:= TRUE);
			p_bytHeaderEnd := strstr(In_pStr:=fbFileRead.pReadBuff,In_pStrSearch:=ADR(FileLc.cTAG_HEADER_E),In_bolAddStrSearchLen:= FALSE);
			IF ((p_bytHeaderBegin=TC3_MEMMAN.NULL) OR (p_bytHeaderEnd=TC3_MEMMAN.NULL) OR (p_bytHeaderBegin>p_bytHeaderEnd)) THEN
				strInfo := CONCAT(STR1:='template/config file: parse error: ',STR2:= FileLc.cTAG_HEADER_B);
				Out_udiStatus := FileLc.cERR_HEADER_TAG;
				RETURN;
			END_IF
			
			// <FOOTER>
			p_bytFooterBegin := strstr(In_pStr:=fbFileRead.pReadBuff,In_pStrSearch:=ADR(FileLc.cTAG_FOOTER_B),In_bolAddStrSearchLen:= TRUE);
			p_bytFooterEnd := strstr(In_pStr:=fbFileRead.pReadBuff,In_pStrSearch:=ADR(FileLc.cTAG_FOOTER_E),In_bolAddStrSearchLen:= FALSE);
			IF ((p_bytFooterBegin=TC3_MEMMAN.NULL) OR (p_bytFooterEnd=TC3_MEMMAN.NULL) OR (p_bytFooterBegin>p_bytFooterEnd)) THEN
				strInfo := CONCAT(STR1:='template/config file: parse error: ',STR2:= FileLc.cTAG_FOOTER_B);
				Out_udiStatus := FileLc.cERR_FOOTER_TAG;
				RETURN;
			END_IF
			
			// <RECORD>
			p_bytRecordBegin := strstr(In_pStr:=fbFileRead.pReadBuff,In_pStrSearch:=ADR(FileLc.cTAG_RECORD_B),In_bolAddStrSearchLen:= TRUE);
			p_bytRecordEnd := strstr(In_pStr:=fbFileRead.pReadBuff,In_pStrSearch:=ADR(FileLc.cTAG_RECORD_E),In_bolAddStrSearchLen:= FALSE);
			IF ((p_bytRecordBegin=TC3_MEMMAN.NULL) OR (p_bytRecordEnd=TC3_MEMMAN.NULL) OR (p_bytRecordBegin>p_bytRecordEnd)) THEN
				strInfo := CONCAT(STR1:='template/config file: parse error: ',STR2:= FileLc.cTAG_RECORD_B);
				Out_udiStatus := FileLc.cERR_RECORD_TAG;
				RETURN;
			END_IF
			
			//*********************************************************	
			// check header
			// allocate memory for header text
			uinTmpLen := UDINT_TO_UINT(p_bytHeaderEnd-p_bytHeaderBegin); // with key words -> len > necessary...
		//test variabel
			MEMSET(destAddr:=pstrTmp,fillByte:=0,n:= SIZEOF(strTmp));
			MEMCPY(destAddr:=pstrTmp,srcAddr:=p_bytHeaderBegin,n:= (SIZEOF(strTmp)-1)); // zero determining string
			
			
			In_pstSysInfo^.p_bytHeaderText := M_AllocMEM(uinTmpLen);
			IF (In_pstSysInfo^.p_bytHeaderText=TC3_MEMMAN.NULL) THEN
				strInfo := 'template/config file: alloc memory for header text failed';
				Out_udiStatus := FileLc.cERR_ALLOC_MEMORY;
				RETURN;
			END_IF
			p_bytTmpDestAdr := In_pstSysInfo^.p_bytHeaderText;
			p_bytTmpSrcAdr := p_bytHeaderBegin;
			uinTmpLen := 0;
			REPEAT
				p_bytRowBegin := strstr(In_pStr:=p_bytTmpSrcAdr,In_pStrSearch:=ADR(FileLc.cTAG_ROW_B),In_bolAddStrSearchLen:= TRUE);
				p_bytRowEnd := strstr(In_pStr:=p_bytTmpSrcAdr,In_pStrSearch:=ADR(FileLc.cTAG_ROW_E),In_bolAddStrSearchLen:= FALSE);
				IF ((p_bytRowBegin<>TC3_MEMMAN.NULL) AND (p_bytRowEnd<>TC3_MEMMAN.NULL) 
					AND (p_bytRowBegin<p_bytHeaderEnd) AND (p_bytRowEnd<p_bytHeaderEnd)) THEN
					IF (p_bytRowBegin>p_bytRowEnd) THEN
						strInfo := CONCAT(STR1:='template/config file: parse error: ',STR2:= FileLc.cTAG_ROW_B);
						strInfo := CONCAT(STR1:=strInfo,STR2:= ' in :');
						strInfo := CONCAT(STR1:=strInfo,STR2:= FileLc.cTAG_HEADER_B);
						Out_udiStatus := FileLc.cERR_ROW_TAG;
						RETURN;
					END_IF
					uinTmpLen := uinTmpLen + DWORD_TO_UINT(p_bytRowEnd-p_bytRowBegin);
					MEMCPY(destAddr:=p_bytTmpDestAdr,srcAddr:=p_bytRowBegin,n:=(p_bytRowEnd-p_bytRowBegin)); // copy row section
			//test variabel
			MEMSET(destAddr:=pstrTmp,fillByte:=0,n:= SIZEOF(strTmp));
			MEMCPY(destAddr:=pstrTmp,srcAddr:=p_bytTmpDestAdr,n:= (SIZEOF(strTmp)-1)); // zero determining string
			
					p_bytTmpDestAdr := p_bytTmpDestAdr + p_bytRowEnd - p_bytRowBegin; //calculate next adress to add texts
					uinTmpLen := uinTmpLen + SIZEOF(FileLc.cEOL);
					MEMCPY(destAddr:=p_bytTmpDestAdr,srcAddr:=ADR(FileLc.cEOL),n:=SIZEOF(FileLc.cEOL)); //add end of line
					p_bytTmpDestAdr := p_bytTmpDestAdr + SIZEOF(FileLc.cEOL);
					p_bytTmpSrcAdr := p_bytRowEnd + Tc2_Standard.LEN(STR:=FileLc.cTAG_ROW_E);
				ELSE
					p_bytRowBegin := TC3_MEMMAN.NULL;
				END_IF
			UNTIL(p_bytRowBegin=TC3_MEMMAN.NULL)
			END_REPEAT
			In_pstSysInfo^.udiHeaderTextLen := UINT_TO_UDINT(uinTmpLen);
			
			
			//*********************************************************	
			// check footer
			// allocate memory for footer text
			uinTmpLen := UDINT_TO_UINT(p_bytFooterEnd-p_bytFooterBegin);// with key words -> len > necessary...
			
			In_pstSysInfo^.p_bytFooterText := M_AllocMEM(uinTmpLen);
			IF (In_pstSysInfo^.p_bytFooterText=TC3_MEMMAN.NULL) THEN
				strInfo := 'template/config file: alloc memory for footer text failed';
				Out_udiStatus := FileLc.cERR_ALLOC_MEMORY;
				RETURN;
			END_IF
			p_bytTmpDestAdr := In_pstSysInfo^.p_bytFooterText;
			p_bytTmpSrcAdr := p_bytFooterBegin;
			uinTmpLen := 0;
			REPEAT
				p_bytRowBegin := strstr(In_pStr:=p_bytTmpSrcAdr,In_pStrSearch:=ADR(FileLc.cTAG_ROW_B),In_bolAddStrSearchLen:= TRUE);
				p_bytRowEnd := strstr(In_pStr:=p_bytTmpSrcAdr,In_pStrSearch:=ADR(FileLc.cTAG_ROW_E),In_bolAddStrSearchLen:= FALSE);
				IF ((p_bytRowBegin<>TC3_MEMMAN.NULL) AND (p_bytRowEnd<>TC3_MEMMAN.NULL) 
					AND (p_bytRowBegin<p_bytFooterEnd) AND (p_bytRowEnd<p_bytFooterEnd)) THEN
					IF (p_bytRowBegin>p_bytRowEnd) THEN
						strInfo := CONCAT(STR1:='template/config file: parse error: ',STR2:= FileLc.cTAG_ROW_B);
						strInfo := CONCAT(STR1:=strInfo,STR2:= ' in :');
						strInfo := CONCAT(STR1:=strInfo,STR2:= FileLc.cTAG_FOOTER_B);
						Out_udiStatus := FileLc.cERR_ROW_TAG;
						RETURN;
					END_IF
					uinTmpLen := uinTmpLen + DWORD_TO_UINT(p_bytRowEnd-p_bytRowBegin);
					MEMCPY(destAddr:=p_bytTmpDestAdr,srcAddr:=p_bytRowBegin,n:=(p_bytRowEnd-p_bytRowBegin)); // copy row section
					p_bytTmpDestAdr := p_bytTmpDestAdr + p_bytRowEnd - p_bytRowBegin; //calculate next adress to add texts
					uinTmpLen := uinTmpLen + SIZEOF(FileLc.cEOL);
					MEMCPY(destAddr:=p_bytTmpDestAdr,srcAddr:=ADR(FileLc.cEOL),n:=SIZEOF(FileLc.cEOL)); //add end of line
					p_bytTmpDestAdr := p_bytTmpDestAdr + SIZEOF(FileLc.cEOL);
					p_bytTmpSrcAdr := p_bytRowEnd + Tc2_Standard.LEN(STR:=FileLc.cTAG_ROW_E);
				ELSE
					p_bytRowBegin := TC3_MEMMAN.NULL;
				END_IF
			UNTIL(p_bytRowBegin=TC3_MEMMAN.NULL)
			END_REPEAT
			In_pstSysInfo^.udiFooterTextLen := UINT_TO_UDINT(uinTmpLen);
			
			//*********************************************************	
			// check RECORD
			uinItemCount := 0;
			p_bytTmpSrcAdr := p_bytRecordBegin;
			
			// count all items in record tag
			REPEAT
				p_bytItemBegin := strstr(In_pStr:=p_bytTmpSrcAdr,In_pStrSearch:=ADR(FileLc.cTAG_ITEM_B),In_bolAddStrSearchLen:= TRUE);
				p_bytItemEnd := strstr(In_pStr:=p_bytTmpSrcAdr,In_pStrSearch:=ADR(FileLc.cTAG_ITEM_E),In_bolAddStrSearchLen:= FALSE);
				
				IF ((p_bytItemBegin<>TC3_MEMMAN.NULL) AND (p_bytItemEnd<>TC3_MEMMAN.NULL) 
					AND (p_bytItemBegin<p_bytRecordEnd) AND (p_bytItemEnd<p_bytRecordEnd)) THEN
					p_bytTmpSrcAdr := p_bytItemEnd + LEN(STR:=FileLc.cTAG_ITEM_E); 
					
					// plausibility check
					IF (p_bytItemBegin>p_bytItemEnd) THEN
						strInfo := CONCAT(STR1:='template/config file: parse error: ',STR2:= FileLc.cTAG_ITEM_B);
						strInfo := CONCAT(STR1:=strInfo,STR2:= ' in :');
						strInfo := CONCAT(STR1:=strInfo,STR2:= FileLc.cTAG_RECORD_B);
						Out_udiStatus := FileLc.cERR_ITEM_TAG;
						RETURN;
					END_IF
					// item tag count
					uinItemCount := uinItemCount +1;
				ELSE
					p_bytItemBegin := TC3_MEMMAN.NULL;
				END_IF
				
			UNTIL(p_bytItemBegin=TC3_MEMMAN.NULL)
			END_REPEAT
			
			// save found number of items
			In_pstSysInfo^.stItemInfo.uinActNbrOfItems := uinItemCount;
			
			// allocate memory for ItemData list
			FOR ii:=0 TO Queue.cMAX_NR_OF_TASKS BY 1 DO
				In_pstSysInfo^.stItemInfo.a_p_bytItemDataList[ii] := M_AllocMEM(uinItemCount*SIZEOF(T_FileLc_ItemData));
				IF (In_pstSysInfo^.stItemInfo.a_p_bytItemDataList[ii]=TC3_MEMMAN.NULL) THEN
					strInfo := 'template/config file: alloc memory for item data list failed';
					Out_udiStatus := FileLc.cERR_ALLOC_MEMORY;
					RETURN;
				END_IF
			END_FOR
			stStatemachine.uinState := stStatemachine.uinState  + 1;
		
		5:
			// allocate memory for ItemCfg list
			In_pstSysInfo^.stItemInfo.p_bytItemCfgList := M_AllocMEM(uinItemCount*SIZEOF(T_FileLc_ItemCfg));
			IF (In_pstSysInfo^.stItemInfo.p_bytItemCfgList=TC3_MEMMAN.NULL) THEN
				strInfo := 'template/config file: alloc memory for item config list failed';
				Out_udiStatus := FileLc.cERR_ALLOC_MEMORY;
				RETURN;
			END_IF
			p_stItemCfgList := In_pstSysInfo^.stItemInfo.p_bytItemCfgList;
			
			//*********************************************************	
			// in RECORD, search all item-tags
			uinItemCount := 0;
			p_bytTmpSrcAdr := p_bytRecordBegin;
			
			// count all items in record tag
			REPEAT
				p_bytItemBegin := strstr(In_pStr:=p_bytTmpSrcAdr,In_pStrSearch:=ADR(FileLc.cTAG_ITEM_B),In_bolAddStrSearchLen:= TRUE);
				p_bytItemEnd := strstr(In_pStr:=p_bytTmpSrcAdr,In_pStrSearch:=ADR(FileLc.cTAG_ITEM_E),In_bolAddStrSearchLen:= FALSE);
				
				IF ((p_bytItemBegin<>TC3_MEMMAN.NULL) AND (p_bytItemEnd<>TC3_MEMMAN.NULL) 
					AND (p_bytItemBegin<p_bytRecordEnd) AND (p_bytItemEnd<p_bytRecordEnd)) THEN
					
					// plausibility check
					IF (p_bytItemBegin>p_bytItemEnd) THEN
						strInfo := CONCAT(STR1:='template/config file: parse error: ',STR2:= FileLc.cTAG_ITEM_B);
						strInfo := CONCAT(STR1:=strInfo,STR2:= ' in :');
						strInfo := CONCAT(STR1:=strInfo,STR2:= FileLc.cTAG_RECORD_B);
						Out_udiStatus := FileLc.cERR_ITEM_TAG;
						RETURN;
					END_IF
					//test variabel
		MEMSET(destAddr:=pstrTmp,fillByte:=0,n:= SIZEOF(strTmp));
		MEMCPY(destAddr:=pstrTmp,srcAddr:=p_bytItemBegin,n:= (SIZEOF(strTmp)-1)); // zero determining string
		
					p_bytTmpSrcAdr := p_bytItemEnd + LEN(STR:=FileLc.cTAG_ITEM_E);
					udiTmpLen := p_bytItemEnd-p_bytItemBegin;
					IF (MEMCMP(pBuf1:=p_bytItemBegin,pBuf2:=ADR(FileLc.cITEM_UNIX_DATE_TIME),udiTmpLen) = 0) THEN
						p_stItemCfgList[uinItemCount].dinPvId := FileLc.cPVTYPE_UNIX_DATE_TIME;		
					ELSIF(MEMCMP(pBuf1:=p_bytItemBegin,pBuf2:=ADR(FileLc.cITEM_UNIX_DATE_TIME_STR),udiTmpLen) = 0) THEN
						p_stItemCfgList[uinItemCount].dinPvId := FileLc.cPVTYPE_UNIX_DATE_TIME_STR;	
					ELSIF(MEMCMP(pBuf1:=p_bytItemBegin,pBuf2:=ADR(FileLc.cITEM_EXCEL_DATE_TIME),udiTmpLen) = 0) THEN
						p_stItemCfgList[uinItemCount].dinPvId := FileLc.cPVTYPE_EXCEL_DATE_TIME;	
					ELSIF(MEMCMP(pBuf1:=p_bytItemBegin,pBuf2:=ADR(FileLc.cITEM_DATE_SLASH_TIME_COLON),udiTmpLen) = 0) THEN
						p_stItemCfgList[uinItemCount].dinPvId := FileLc.cPVTYPE_DATE_SLASH_TIME_COLON;		
					ELSIF(MEMCMP(pBuf1:=p_bytItemBegin,pBuf2:=ADR(FileLc.cITEM_TIME_MILLI),udiTmpLen) = 0) THEN
						p_stItemCfgList[uinItemCount].dinPvId := FileLc.cPVTYPE_TIME_MILLI;	
					ELSIF(MEMCMP(pBuf1:=p_bytItemBegin,pBuf2:=ADR(FileLc.cITEM_BL_LOGTYP),udiTmpLen) = 0) THEN
						p_stItemCfgList[uinItemCount].dinPvId := FileLc.cPVTYPE_BL_LOGTYP;	
					ELSIF(MEMCMP(pBuf1:=p_bytItemBegin,pBuf2:=ADR(FileLc.cITEM_BL_CTRL_ID),udiTmpLen) = 0) THEN
						p_stItemCfgList[uinItemCount].dinPvId := FileLc.cPVTYPE_BL_CTRL_ID;	
					ELSIF(MEMCMP(pBuf1:=p_bytItemBegin,pBuf2:=ADR(FileLc.cITEM_BL_STRING1),udiTmpLen) = 0) THEN
						p_stItemCfgList[uinItemCount].dinPvId := FileLc.cPVTYPE_BL_STRING1;	
					ELSIF(MEMCMP(pBuf1:=p_bytItemBegin,pBuf2:=ADR(FileLc.cITEM_BL_STRING2),udiTmpLen) = 0) THEN
						p_stItemCfgList[uinItemCount].dinPvId := FileLc.cPVTYPE_BL_STRING2;	
					ELSIF(MEMCMP(pBuf1:=p_bytItemBegin,pBuf2:=ADR(FileLc.cITEM_BL_PAR1),udiTmpLen) = 0) THEN
						p_stItemCfgList[uinItemCount].dinPvId := FileLc.cPVTYPE_BL_PAR1;	
					ELSIF(MEMCMP(pBuf1:=p_bytItemBegin,pBuf2:=ADR(FileLc.cITEM_BL_PAR2),udiTmpLen) = 0) THEN
						p_stItemCfgList[uinItemCount].dinPvId := FileLc.cPVTYPE_BL_PAR2;
					ELSIF(MEMCMP(pBuf1:=p_bytItemBegin,pBuf2:=ADR(FileLc.cITEM_BL_PAR3),udiTmpLen) = 0) THEN
						p_stItemCfgList[uinItemCount].dinPvId := FileLc.cPVTYPE_BL_PAR3;
					ELSIF(MEMCMP(pBuf1:=p_bytItemBegin,pBuf2:=ADR(FileLc.cITEM_BL_PAR4),udiTmpLen) = 0) THEN
						p_stItemCfgList[uinItemCount].dinPvId := FileLc.cPVTYPE_BL_PAR4;
					ELSE
						MEMSET(destAddr := ADR(strTmp),0,SIZEOF(strTmp));
						IF (udiTmpLen < SIZEOF(strTmp)) THEN
							MEMCPY(destAddr := ADR(strTmp),srcAddr := p_bytItemBegin,udiTmpLen);
							p_stItemCfgList[uinItemCount].dinPvId := STRING_TO_DINT(strTmp);
						ELSE
							strInfo := CONCAT(STR1:='template/config file: parse error item definition larger than defined string: ',STR2:= FileLc.cTAG_ITEM_B);
							strInfo := CONCAT(STR1:=strInfo,STR2:= ' in :');
							strInfo := CONCAT(STR1:=strInfo,STR2:= FileLc.cTAG_RECORD_B);
							Out_udiStatus := FileLc.cERR_ITEM_TAG;
							RETURN;
						END_IF
					END_IF
					
					IF (uinItemCount=0) THEN // only for the first element
						// PreText
						udiTmpLen := p_bytItemBegin-Tc2_Standard.LEN(STR:=FileLc.cTAG_ITEM_B)-p_bytRecordBegin;
						IF (udiTmpLen>FileLc.cPRE_POST_TEXTLEN) THEN
							udiTmpLen := FileLc.cPRE_POST_TEXTLEN - 1; //-1 -> strEnd!
						END_IF
						MEMSET(destAddr := ADR(In_pstSysInfo^.stItemInfo.strPreItemText),0,SIZEOF(In_pstSysInfo^.stItemInfo.strPreItemText));
						MEMCPY(destAddr:=ADR(In_pstSysInfo^.stItemInfo.strPreItemText), p_bytRecordBegin, udiTmpLen);
					ELSE
						// Post item text
						udiTmpLen := p_bytItemBegin-Tc2_Standard.LEN(STR:=FileLc.cTAG_ITEM_B)-p_bytLastPos;
						IF (udiTmpLen>FileLc.cPRE_POST_TEXTLEN) THEN
							udiTmpLen := FileLc.cPRE_POST_TEXTLEN - 1; //-1 -> strEnd!
						END_IF
						MEMSET(destAddr := ADR(p_stItemCfgList[uinItemCount-1].strPostText),0,SIZEOF(p_stItemCfgList[uinItemCount-1].strPostText));
						MEMCPY(destAddr:=ADR(p_stItemCfgList[uinItemCount-1].strPostText), p_bytLastPos, udiTmpLen);
					END_IF
					
					// save last position of ITEM entry
					p_bytLastPos := p_bytItemEnd + Tc2_Standard.LEN(STR:=FileLc.cTAG_ITEM_E);
					// item tag count
					uinItemCount := uinItemCount +1;
				ELSE
					p_bytItemBegin := TC3_MEMMAN.NULL;
				END_IF
				
			UNTIL(p_bytItemBegin=TC3_MEMMAN.NULL)
			END_REPEAT
			
			// manage last element
			udiTmpLen := p_bytRecordEnd-p_bytLastPos;
			IF (udiTmpLen>FileLc.cPRE_POST_TEXTLEN) THEN
				udiTmpLen := FileLc.cPRE_POST_TEXTLEN - 1; //-1 -> strEnd!
			END_IF
			MEMCPY(destAddr:=ADR(p_stItemCfgList[uinItemCount-1].strPostText), p_bytLastPos, udiTmpLen);
			
			//*********************************************************	
			// check CONFIG 
			
			//**** <LOGFILE_PRAEFIX>
			p_bytConfigValBegin := strstr(In_pStr:=p_bytConfigBegin,In_pStrSearch:=ADR(FileLc.cTAG_CFG_LOGFILE_PRAEFIX_B),In_bolAddStrSearchLen:= TRUE);
			p_bytConfigValEnd := strstr(In_pStr:=p_bytConfigBegin,In_pStrSearch:=ADR(FileLc.cTAG_CFG_LOGFILE_PRAEFIX_E),In_bolAddStrSearchLen:= FALSE);
			IF ((p_bytConfigValBegin<>TC3_MEMMAN.NULL) AND (p_bytConfigValEnd<>TC3_MEMMAN.NULL) AND (p_bytConfigValBegin<p_bytConfigValEnd) AND (p_bytConfigValEnd<p_bytConfigEnd)) THEN
				MEMSET(destAddr := ADR(strTmp),0,SIZEOF(strTmp));
				udiTmpLen := p_bytConfigValEnd - p_bytConfigValBegin;
		
				IF (SIZEOF(strTmp)>udiTmpLen) THEN
					MEMCPY(destAddr := ADR(strTmp),srcAddr := p_bytConfigValBegin,udiTmpLen);	
				ELSE
					strTmp := FileLc.cCFG_LOGFILE_NAME; // error - load default
				END_IF
			ELSE
				strTmp := FileLc.cCFG_LOGFILE_NAME; // error - load default
			END_IF
			In_pstSysInfo^.stConfig.strLogFileNamePraeFix := strTmp;
			
			//**** <LOGFILE_EXT>
			p_bytConfigValBegin := strstr(In_pStr:=p_bytConfigBegin,In_pStrSearch:=ADR(FileLc.cTAG_CFG_LOGFILE_EXT_B),In_bolAddStrSearchLen:= TRUE);
			p_bytConfigValEnd := strstr(In_pStr:=p_bytConfigBegin,In_pStrSearch:=ADR(FileLc.cTAG_CFG_LOGFILE_EXT_E),In_bolAddStrSearchLen:= FALSE);
			IF ((p_bytConfigValBegin<>TC3_MEMMAN.NULL) AND (p_bytConfigValEnd<>TC3_MEMMAN.NULL) AND (p_bytConfigValBegin<p_bytConfigValEnd) AND (p_bytConfigValEnd<p_bytConfigEnd)) THEN
				MEMSET(destAddr := ADR(strTmp),0,SIZEOF(strTmp));
				udiTmpLen := p_bytConfigValEnd - p_bytConfigValBegin;
		
				IF (SIZEOF(strTmp)>udiTmpLen) THEN
					MEMCPY(destAddr := ADR(strTmp),srcAddr := p_bytConfigValBegin,udiTmpLen);	
				ELSE
					strTmp := FileLc.cCFG_LOGFILE_EXT; // error - load default
				END_IF
			ELSE
				strTmp := FileLc.cCFG_LOGFILE_EXT; // error - load default
			END_IF
			In_pstSysInfo^.stConfig.strLogFileNameExt := strTmp;
			
			//**** <LOG_TIMESTAMP>
			
			p_bytConfigValBegin := strstr(In_pStr:=p_bytConfigBegin,In_pStrSearch:=ADR(FileLc.cTAG_CFG_LOG_TIMESTAMP_B),In_bolAddStrSearchLen:= TRUE);
			p_bytConfigValEnd := strstr(In_pStr:=p_bytConfigBegin,In_pStrSearch:=ADR(FileLc.cTAG_CFG_LOG_TIMESTAMP_E),In_bolAddStrSearchLen:= FALSE);
			IF ((p_bytConfigValBegin<>TC3_MEMMAN.NULL) AND (p_bytConfigValEnd<>TC3_MEMMAN.NULL) AND (p_bytConfigValBegin<p_bytConfigValEnd) AND (p_bytConfigValEnd<p_bytConfigEnd)) THEN
				MEMSET(destAddr := ADR(strTmp),0,SIZEOF(strTmp));
				udiTmpLen := p_bytConfigValEnd - p_bytConfigValBegin;
		
				IF (SIZEOF(strTmp)>udiTmpLen) THEN
					MEMCPY(destAddr := ADR(strTmp),srcAddr := p_bytConfigValBegin,udiTmpLen);	
					IF (FIND(STR1:=strTmp,STR2:=FileLc.cLOG_TIMESTAMP_WIN)<>0)THEN // win defiend
						bolTmp := TRUE;
					ELSE
						bolTmp := FALSE;
					END_IF
				ELSE
					bolTmp := FALSE; // error - load default - local drive access
				END_IF
			ELSE
				bolTmp := FALSE; // error - load default - local drive access
			END_IF
			In_pstSysInfo^.stConfig.bolUseLocalTimeStamp := bolTmp;
			
			//**** <LOGFILE_SNETID>
			p_bytConfigValBegin := strstr(In_pStr:=p_bytConfigBegin,In_pStrSearch:=ADR(FileLc.cTAG_CFG_LOGFILE_SNETID_B),In_bolAddStrSearchLen:= TRUE);
			p_bytConfigValEnd := strstr(In_pStr:=p_bytConfigBegin,In_pStrSearch:=ADR(FileLc.cTAG_CFG_LOGFILE_SNETID_E),In_bolAddStrSearchLen:= FALSE);
			IF ((p_bytConfigValBegin<>TC3_MEMMAN.NULL) AND (p_bytConfigValEnd<>TC3_MEMMAN.NULL) AND (p_bytConfigValBegin<p_bytConfigValEnd) AND (p_bytConfigValEnd<p_bytConfigEnd)) THEN
				MEMSET(destAddr := ADR(strTmp),0,SIZEOF(strTmp));
				udiTmpLen := p_bytConfigValEnd - p_bytConfigValBegin;
		
				IF (SIZEOF(strTmp)>udiTmpLen) THEN
					MEMCPY(destAddr := ADR(strTmp),srcAddr := p_bytConfigValBegin,udiTmpLen);	
				ELSE
					strTmp := ''; // error - load default - local drive access
				END_IF
			ELSE
				strTmp :=  ''; // error - load default - local drive access
			END_IF
			In_pstSysInfo^.stConfig.strLogNetId := strTmp;
			
			//**** <LOGFILE_PATH>
			p_bytConfigValBegin := strstr(In_pStr:=p_bytConfigBegin,In_pStrSearch:=ADR(FileLc.cTAG_CFG_LOGFILE_PATH_B),In_bolAddStrSearchLen:= TRUE);
			p_bytConfigValEnd := strstr(In_pStr:=p_bytConfigBegin,In_pStrSearch:=ADR(FileLc.cTAG_CFG_LOGFILE_PATH_E),In_bolAddStrSearchLen:= FALSE);
			IF ((p_bytConfigValBegin<>TC3_MEMMAN.NULL) AND (p_bytConfigValEnd<>TC3_MEMMAN.NULL) AND (p_bytConfigValBegin<p_bytConfigValEnd) AND (p_bytConfigValEnd<p_bytConfigEnd)) THEN
				MEMSET(destAddr := ADR(strTmp),0,SIZEOF(strTmp));
				udiTmpLen := p_bytConfigValEnd - p_bytConfigValBegin;
		
				IF (SIZEOF(strTmp)>udiTmpLen) THEN
					MEMCPY(destAddr := ADR(strTmp),srcAddr := p_bytConfigValBegin,udiTmpLen);	
				ELSE
					strTmp := In_strPath; // error - load default
				END_IF
			ELSE
				strTmp := In_strPath; // error - load default
			END_IF
			In_pstSysInfo^.stConfig.strLogPath := CONCAT(STR1:=strTmp ,STR2:= '\');
			
			//**** <QEUE_LEN>
			p_bytConfigValBegin := strstr(In_pStr:=p_bytConfigBegin,In_pStrSearch:=ADR(FileLc.cTAG_CFG_QUEUE_LEN_B),In_bolAddStrSearchLen:= TRUE);
			p_bytConfigValEnd := strstr(In_pStr:=p_bytConfigBegin,In_pStrSearch:=ADR(FileLc.cTAG_CFG_QUEUE_LEN_E),In_bolAddStrSearchLen:= FALSE);
			IF ((p_bytConfigValBegin<>TC3_MEMMAN.NULL) AND (p_bytConfigValEnd<>TC3_MEMMAN.NULL) AND (p_bytConfigValBegin<p_bytConfigValEnd) AND (p_bytConfigValEnd<p_bytConfigEnd)) THEN
				MEMSET(destAddr := ADR(strTmp),0,SIZEOF(strTmp));
				udiTmpLen := p_bytConfigValEnd - p_bytConfigValBegin;
		
				IF (SIZEOF(strTmp)>udiTmpLen) THEN
					MEMCPY(destAddr := ADR(strTmp),srcAddr := p_bytConfigValBegin,udiTmpLen);	
					In_pstSysInfo^.stConfig.udiQueueLen := STRING_TO_UDINT(strTmp);
				ELSE
					In_pstSysInfo^.stConfig.udiQueueLen := FileLc.cCFG_QUEUE_LEN; // error - load default
				END_IF
			ELSE
				In_pstSysInfo^.stConfig.udiQueueLen := FileLc.cCFG_QUEUE_LEN; // error - load default
			END_IF
			
